LIN {X 0,Y 213.734,Z 203.361,A -85,B 0,C 180,E1 -20828.664,E2 -20828.664} C_VEL
LIN {X 0,Y 213.771,Z 203.358,A -85,B 0,C 180,E1 -20833.676,E2 -20833.676} C_VEL
LIN {X 0,Y 213.726,Z 203.362,A -85,B 0,C 180,E1 -20836.337,E2 -20836.337} C_VEL
LIN {X 0,Y 213.733,Z 203.362,A -85,B 0,C 180,E1 -20841.337,E2 -20841.337} C_VEL
LIN {X 0,Y 213.765,Z 203.356,A -85,B 0,C 180,E1 -20846.021,E2 -20846.021} C_VEL
LIN {X 0,Y 213.777,Z 203.356,A -85,B 0,C 180,E1 -20850.455,E2 -20850.455} C_VEL
LIN {X 0,Y 213.798,Z 203.348,A -85,B 0,C 180,E1 -20854.702,E2 -20854.702} C_VEL
LIN {X 0,Y 213.809,Z 203.349,A -85,B 0,C 180,E1 -20858.804,E2 -20858.804} C_VEL
LIN {X 0,Y 213.94,Z 203.337,A -85,B 0,C 180,E1 -20862.804,E2 -20862.804} C_VEL
LIN {X 0,Y 213.95,Z 203.333,A -85,B 0,C 180,E1 -20866.707,E2 -20866.707} C_VEL
LIN {X 0,Y 214.139,Z 203.305,A -85,B 0,C 180,E1 -20870.556,E2 -20870.556} C_VEL
LIN {X 0,Y 214.096,Z 203.312,A -85,B 0,C 180,E1 -20874.349,E2 -20874.349} C_VEL
LIN {X 0,Y 214.441,Z 203.245,A -85,B 0,C 180,E1 -20878.123,E2 -20878.123} C_VEL
LIN {X 0,Y 214.547,Z 203.245,A -85,B 0,C 180,E1 -20880.001,E2 -20880.001} C_VEL
LIN {X 0,Y 214.442,Z 203.27,A -85,B 0,C 180,E1 -20881.879,E2 -20881.879} C_VEL
LIN {X 0,Y 214.196,Z 203.304,A -85,B 0,C 180,E1 -20887.543,E2 -20887.543} C_VEL
LIN {X 0,Y 213.997,Z 203.329,A -85,B 0,C 180,E1 -20891.365,E2 -20891.365} C_VEL
LIN {X 0,Y 213.931,Z 203.337,A -85,B 0,C 180,E1 -20895.238,E2 -20895.238} C_VEL
LIN {X 0,Y 213.839,Z 203.349,A -85,B 0,C 180,E1 -20899.188,E2 -20899.188} C_VEL
LIN {X 0,Y 213.847,Z 203.35,A -85,B 0,C 180,E1 -20903.228,E2 -20903.228} C_VEL
LIN {X 0,Y 213.862,Z 203.711,A -85,B 0,C 180,E1 -20907.393,E2 -20907.393} C_VEL
LIN {X 0,Y 214.057,Z 205.405,A -85,B 0,C 180,E1 -20911.691,E2 -20911.691} C_VEL
LIN {X 0,Y 214.298,Z 207.41,A -85,B 0,C 180,E1 -20916.181,E2 -20916.181} C_VEL
LIN {X 0,Y 214.668,Z 209.889,A -85,B 0,C 180,E1 -20921.15,E2 -20921.15} C_VEL
LIN {X 0,Y 214.851,Z 211.419,A -85,B 0,C 180,E1 -20923.976,E2 -20923.976} C_VEL
LIN {X 0,Y 214.879,Z 212.962,A -85,B 0,C 180,E1 -20926.62,E2 -20926.62} C_VEL
LIN {X 0,Y 214.729,Z 214.501,A -85,B 0,C 180,E1 -20929.112,E2 -20929.112} C_VEL
LIN {X 0,Y 213.905,Z 217.533,A -85,B 0,C 180,E1 -20933.744,E2 -20933.744} C_VEL
LIN {X 0,Y 213.736,Z 218.183,A -85,B 0,C 180,E1 -20934.657,E2 -20934.657} C_VEL
LIN {X 0,Y 214.709,Z 221.629,A -85,B 0,C 180,E1 -20935.032,E2 -20935.032} C_VEL
LIN {X 0,Y 218.172,Z 231.953,A -85,B 0,C 180,E1 -20936.447,E2 -20936.447} C_VEL
LIN {X 0,Y 221.362,Z 245.09,A -85,B 0,C 180,E1 -20938.386,E2 -20938.386} C_VEL
LIN {X 0,Y 223.043,Z 255.539,A -85,B 0,C 180,E1 -20940.087,E2 -20940.087} C_VEL
LIN {X 0,Y 223.802,Z 263.81,A -85,B 0,C 180,E1 -20941.557,E2 -20941.557} C_VEL
LIN {X 0,Y 223.987,Z 273.301,A -85,B 0,C 180,E1 -20943.443,E2 -20943.443} C_VEL
LIN {X 0,Y 223.651,Z 277.858,A -85,B 0,C 180,E1 -20944.401,E2 -20944.401} C_VEL
LIN {X 0,Y 220.772,Z 288.296,A -85,B 0,C 180,E1 -20946.813,E2 -20946.813} C_VEL
LIN {X 0,Y 218.78,Z 295.491,A -85,B 0,C 180,E1 -20948.892,E2 -20948.892} C_VEL
LIN {X 0,Y 216.831,Z 301.814,A -85,B 0,C 180,E1 -20951.088,E2 -20951.088} C_VEL
LIN {X 0,Y 215.383,Z 306.725,A -85,B 0,C 180,E1 -20953.129,E2 -20953.129} C_VEL
LIN {X 0,Y 213.86,Z 309.596,A -85,B 0,C 180,E1 -20954.466,E2 -20954.466} C_VEL
LIN {X 0,Y 209.854,Z 313.608,A -85,B 0,C 180,E1 -20956.656,E2 -20956.656} C_VEL
LIN {X 0,Y 206.095,Z 317.034,A -85,B 0,C 180,E1 -20959.002,E2 -20959.002} C_VEL
LIN {X 0,Y 204.99,Z 318.689,A -85,B 0,C 180,E1 -20960.554,E2 -20960.554} C_VEL
LIN {X 0,Y 204.442,Z 321.502,A -85,B 0,C 180,E1 -20964.081,E2 -20964.081} C_VEL
LIN {X 0,Y 204.339,Z 322.566,A -85,B 0,C 180,E1 -20966.056,E2 -20966.056} C_VEL
LIN {X 0,Y 204.365,Z 323.161,A -85,B 0,C 180,E1 -20968.029,E2 -20968.029} C_VEL
LIN {X 0,Y 204.429,Z 323.319,A -85,B 0,C 180,E1 -20970,E2 -20970} C_VEL
LIN {X 0,Y 204.366,Z 323.161,A -85,B 0,C 180,E1 -20971.971,E2 -20971.971} C_VEL
LIN {X 0,Y 204.36,Z 322.491,A -85,B 0,C 180,E1 -20974.184,E2 -20974.184} C_VEL
LIN {X 0,Y 204.675,Z 320.109,A -85,B 0,C 180,E1 -20977.894,E2 -20977.894} C_VEL
LIN {X 0,Y 205.363,Z 317.152,A -85,B 0,C 180,E1 -20980.849,E2 -20980.849} C_VEL
LIN {X 0,Y 206.412,Z 313.156,A -85,B 0,C 180,E1 -20983.788,E2 -20983.788} C_VEL
LIN {X 0,Y 208.044,Z 308.023,A -85,B 0,C 180,E1 -20986.687,E2 -20986.687} C_VEL
LIN {X 0,Y 209.717,Z 302.758,A -85,B 0,C 180,E1 -20989.071,E2 -20989.071} C_VEL
LIN {X 0,Y 211.811,Z 296.441,A -85,B 0,C 180,E1 -20991.406,E2 -20991.406} C_VEL
LIN {X 0,Y 213.493,Z 290.484,A -85,B 0,C 180,E1 -20993.267,E2 -20993.267} C_VEL
LIN {X 0,Y 215.527,Z 283.556,A -85,B 0,C 180,E1 -20995.081,E2 -20995.081} C_VEL
LIN {X 0,Y 217.216,Z 277.645,A -85,B 0,C 180,E1 -20996.415,E2 -20996.415} C_VEL
LIN {X 0,Y 217.345,Z 267.824,A -85,B 0,C 180,E1 -20998.547,E2 -20998.547} C_VEL
LIN {X 0,Y 216.74,Z 258.58,A -85,B 0,C 180,E1 -21000.341,E2 -21000.341} C_VEL
LIN {X 0,Y 215.465,Z 249.191,A -85,B 0,C 180,E1 -21001.997,E2 -21001.997} C_VEL
LIN {X 0,Y 213.303,Z 238.611,A -85,B 0,C 180,E1 -21003.699,E2 -21003.699} C_VEL
LIN {X 0,Y 210.592,Z 229.072,A -85,B 0,C 180,E1 -21005.149,E2 -21005.149} C_VEL
LIN {X 0,Y 207.683,Z 220.968,A -85,B 0,C 180,E1 -21006.358,E2 -21006.358} C_VEL
LIN {X 0,Y 206.902,Z 217.966,A -85,B 0,C 180,E1 -21006.726,E2 -21006.726} C_VEL
LIN {X 0,Y 207.478,Z 215.775,A -85,B 0,C 180,E1 -21010.06,E2 -21010.06} C_VEL
LIN {X 0,Y 207.75,Z 214.247,A -85,B 0,C 180,E1 -21012.576,E2 -21012.576} C_VEL
LIN {X 0,Y 207.807,Z 212.729,A -85,B 0,C 180,E1 -21015.252,E2 -21015.252} C_VEL
LIN {X 0,Y 207.52,Z 210.25,A -85,B 0,C 180,E1 -21019.948,E2 -21019.948} C_VEL
LIN {X 0,Y 207.225,Z 207.973,A -85,B 0,C 180,E1 -21024.79,E2 -21024.79} C_VEL
LIN {X 0,Y 206.981,Z 206.053,A -85,B 0,C 180,E1 -21029.38,E2 -21029.38} C_VEL
LIN {X 0,Y 206.751,Z 204.425,A -85,B 0,C 180,E1 -21033.774,E2 -21033.774} C_VEL
LIN {X 0,Y 206.757,Z 204.236,A -85,B 0,C 180,E1 -21038.042,E2 -21038.042} C_VEL
LIN {X 0,Y 206.873,Z 204.219,A -85,B 0,C 180,E1 -21042.195,E2 -21042.195} C_VEL
LIN {X 0,Y 206.893,Z 204.215,A -85,B 0,C 180,E1 -21046.243,E2 -21046.243} C_VEL
LIN {X 0,Y 207.098,Z 204.19,A -85,B 0,C 180,E1 -21050.23,E2 -21050.23} C_VEL
LIN {X 0,Y 207.058,Z 204.194,A -85,B 0,C 180,E1 -21054.155,E2 -21054.155} C_VEL
LIN {X 0,Y 207.378,Z 204.15,A -85,B 0,C 180,E1 -21058.057,E2 -21058.057} C_VEL
LIN {X 0,Y 207.512,Z 204.12,A -85,B 0,C 180,E1 -21059.999,E2 -21059.999} C_VEL
LIN {X 0,Y 207.378,Z 204.124,A -85,B 0,C 180,E1 -21061.941,E2 -21061.941} C_VEL
LIN {X 0,Y 207.138,Z 204.182,A -85,B 0,C 180,E1 -21067.799,E2 -21067.799} C_VEL
LIN {X 0,Y 206.928,Z 204.21,A -85,B 0,C 180,E1 -21071.757,E2 -21071.757} C_VEL
LIN {X 0,Y 206.863,Z 204.214,A -85,B 0,C 180,E1 -21075.77,E2 -21075.77} C_VEL
LIN {X 0,Y 206.78,Z 204.219,A -85,B 0,C 180,E1 -21079.868,E2 -21079.868} C_VEL
LIN {X 0,Y 206.76,Z 204.227,A -85,B 0,C 180,E1 -21084.071,E2 -21084.071} C_VEL
LIN {X 0,Y 206.741,Z 204.233,A -85,B 0,C 180,E1 -21088.418,E2 -21088.418} C_VEL
LIN {X 0,Y 206.705,Z 204.236,A -85,B 0,C 180,E1 -21092.955,E2 -21092.955} C_VEL
LIN {X 0,Y 206.718,Z 204.234,A -85,B 0,C 180,E1 -21095.32,E2 -21095.32} C_VEL
LIN {X 0,Y 206.667,Z 204.242,A -85,B 0,C 180,E1 -21100.248,E2 -21100.248} C_VEL
LIN {X 0,Y 206.645,Z 204.245,A -85,B 0,C 180,E1 -21104.422,E2 -21104.422} C_VEL
LIN {X 0,Y 206.659,Z 204.241,A -85,B 0,C 180,E1 -21109.749,E2 -21109.749} C_VEL
LIN {X 0,Y 206.695,Z 204.302,A -85,B 0,C 180,E1 -21113.054,E2 -21113.054} C_VEL
LIN {X 0,Y 207.675,Z 207.027,A -85,B 0,C 180,E1 -21113.414,E2 -21113.414} C_VEL
LIN {X 0,Y 209.169,Z 209.299,A -85,B 0,C 180,E1 -21113.848,E2 -21113.848} C_VEL
LIN {X 0,Y 214.287,Z 218.562,A -85,B 0,C 180,E1 -21115.53,E2 -21115.53} C_VEL
LIN {X 0,Y 219.411,Z 229.769,A -85,B 0,C 180,E1 -21117.559,E2 -21117.559} C_VEL
LIN {X 0,Y 223.293,Z 240.321,A -85,B 0,C 180,E1 -21119.548,E2 -21119.548} C_VEL
LIN {X 0,Y 226.869,Z 250.975,A -85,B 0,C 180,E1 -21121.781,E2 -21121.781} C_VEL
LIN {X 0,Y 230.64,Z 259.099,A -85,B 0,C 180,E1 -21123.821,E2 -21123.821} C_VEL
LIN {X 0,Y 235.944,Z 267.711,A -85,B 0,C 180,E1 -21126.336,E2 -21126.336} C_VEL
LIN {X 0,Y 242.815,Z 276.218,A -85,B 0,C 180,E1 -21129.203,E2 -21129.203} C_VEL
LIN {X 0,Y 250.96,Z 283.988,A -85,B 0,C 180,E1 -21132.201,E2 -21132.201} C_VEL
LIN {X 0,Y 258.511,Z 290.027,A -85,B 0,C 180,E1 -21134.816,E2 -21134.816} C_VEL
LIN {X 0,Y 267.698,Z 296.215,A -85,B 0,C 180,E1 -21137.876,E2 -21137.876} C_VEL
LIN {X 0,Y 274.849,Z 300.626,A -85,B 0,C 180,E1 -21140.433,E2 -21140.433} C_VEL
LIN {X 0,Y 280.845,Z 303.994,A -85,B 0,C 180,E1 -21142.812,E2 -21142.812} C_VEL
LIN {X 0,Y 283.79,Z 305.702,A -85,B 0,C 180,E1 -21144.315,E2 -21144.315} C_VEL
LIN {X 0,Y 285.961,Z 307.015,A -85,B 0,C 180,E1 -21145.772,E2 -21145.772} C_VEL
LIN {X 0,Y 288.415,Z 308.115,A -85,B 0,C 180,E1 -21147.514,E2 -21147.514} C_VEL
LIN {X 0,Y 289.581,Z 308.494,A -85,B 0,C 180,E1 -21148.609,E2 -21148.609} C_VEL
LIN {X 0,Y 290.591,Z 308.662,A -85,B 0,C 180,E1 -21150,E2 -21150} C_VEL
LIN {X 0,Y 289.596,Z 308.494,A -85,B 0,C 180,E1 -21151.391,E2 -21151.391} C_VEL
LIN {X 0,Y 287.978,Z 307.95,A -85,B 0,C 180,E1 -21152.798,E2 -21152.798} C_VEL
LIN {X 0,Y 285.97,Z 307.014,A -85,B 0,C 180,E1 -21154.228,E2 -21154.228} C_VEL
LIN {X 0,Y 282.805,Z 305.083,A -85,B 0,C 180,E1 -21156.266,E2 -21156.266} C_VEL
LIN {X 0,Y 280.814,Z 303.995,A -85,B 0,C 180,E1 -21157.189,E2 -21157.189} C_VEL
LIN {X 0,Y 274.935,Z 300.623,A -85,B 0,C 180,E1 -21159.564,E2 -21159.564} C_VEL
LIN {X 0,Y 267.713,Z 296.215,A -85,B 0,C 180,E1 -21162.123,E2 -21162.123} C_VEL
LIN {X 0,Y 258.512,Z 290.025,A -85,B 0,C 180,E1 -21165.185,E2 -21165.185} C_VEL
LIN {X 0,Y 250.459,Z 283.545,A -85,B 0,C 180,E1 -21167.978,E2 -21167.978} C_VEL
LIN {X 0,Y 242.837,Z 276.198,A -85,B 0,C 180,E1 -21170.8,E2 -21170.8} C_VEL
LIN {X 0,Y 235.921,Z 267.776,A -85,B 0,C 180,E1 -21173.651,E2 -21173.651} C_VEL
LIN {X 0,Y 230.036,Z 257.992,A -85,B 0,C 180,E1 -21176.481,E2 -21176.481} C_VEL
LIN {X 0,Y 225.736,Z 248.075,A -85,B 0,C 180,E1 -21178.874,E2 -21178.874} C_VEL
LIN {X 0,Y 222.35,Z 237.621,A -85,B 0,C 180,E1 -21180.963,E2 -21180.963} C_VEL
LIN {X 0,Y 219.407,Z 229.775,A -85,B 0,C 180,E1 -21182.441,E2 -21182.441} C_VEL
LIN {X 0,Y 214.208,Z 218.418,A -85,B 0,C 180,E1 -21184.497,E2 -21184.497} C_VEL
LIN {X 0,Y 208.571,Z 208.219,A -85,B 0,C 180,E1 -21186.356,E2 -21186.356} C_VEL
LIN {X 0,Y 207.015,Z 205.604,A -85,B 0,C 180,E1 -21186.82,E2 -21186.82} C_VEL
LIN {X 0,Y 206.689,Z 204.239,A -85,B 0,C 180,E1 -21187.018,E2 -21187.018} C_VEL
LIN {X 0,Y 206.675,Z 204.242,A -85,B 0,C 180,E1 -21191.575,E2 -21191.575} C_VEL
LIN {X 0,Y 206.648,Z 204.244,A -85,B 0,C 180,E1 -21195.577,E2 -21195.577} C_VEL
LIN {X 0,Y 206.667,Z 204.242,A -85,B 0,C 180,E1 -21199.752,E2 -21199.752} C_VEL
LIN {X 0,Y 206.728,Z 204.233,A -85,B 0,C 180,E1 -21204.696,E2 -21204.696} C_VEL
LIN {X 0,Y 206.72,Z 204.235,A -85,B 0,C 180,E1 -21209.34,E2 -21209.34} C_VEL
LIN {X 0,Y 206.729,Z 204.23,A -85,B 0,C 180,E1 -21213.773,E2 -21213.773} C_VEL
LIN {X 0,Y 206.754,Z 204.23,A -85,B 0,C 180,E1 -21218.044,E2 -21218.044} C_VEL
LIN {X 0,Y 206.87,Z 204.216,A -85,B 0,C 180,E1 -21222.197,E2 -21222.197} C_VEL
LIN {X 0,Y 206.892,Z 204.21,A -85,B 0,C 180,E1 -21226.245,E2 -21226.245} C_VEL
LIN {X 0,Y 207.097,Z 204.182,A -85,B 0,C 180,E1 -21230.232,E2 -21230.232} C_VEL
LIN {X 0,Y 207.058,Z 204.191,A -85,B 0,C 180,E1 -21234.157,E2 -21234.157} C_VEL
LIN {X 0,Y 207.378,Z 204.124,A -85,B 0,C 180,E1 -21238.059,E2 -21238.059} C_VEL
LIN {X 0,Y 207.512,Z 204.12,A -85,B 0,C 180,E1 -21240.001,E2 -21240.001} C_VEL
LIN {X 0,Y 207.378,Z 204.15,A -85,B 0,C 180,E1 -21241.943,E2 -21241.943} C_VEL
LIN {X 0,Y 207.138,Z 204.184,A -85,B 0,C 180,E1 -21247.801,E2 -21247.801} C_VEL
LIN {X 0,Y 206.923,Z 204.212,A -85,B 0,C 180,E1 -21251.76,E2 -21251.76} C_VEL
LIN {X 0,Y 206.865,Z 204.219,A -85,B 0,C 180,E1 -21255.772,E2 -21255.772} C_VEL
LIN {X 0,Y 206.783,Z 204.229,A -85,B 0,C 180,E1 -21259.87,E2 -21259.87} C_VEL
LIN {X 0,Y 206.763,Z 204.231,A -85,B 0,C 180,E1 -21264.073,E2 -21264.073} C_VEL
LIN {X 0,Y 206.751,Z 204.419,A -85,B 0,C 180,E1 -21266.226,E2 -21266.226} C_VEL
LIN {X 0,Y 206.981,Z 206.052,A -85,B 0,C 180,E1 -21270.62,E2 -21270.62} C_VEL
LIN {X 0,Y 207.238,Z 208.124,A -85,B 0,C 180,E1 -21275.522,E2 -21275.522} C_VEL
LIN {X 0,Y 207.526,Z 210.283,A -85,B 0,C 180,E1 -21280.051,E2 -21280.051} C_VEL
LIN {X 0,Y 207.807,Z 212.733,A -85,B 0,C 180,E1 -21284.748,E2 -21284.748} C_VEL
LIN {X 0,Y 207.711,Z 214.682,A -85,B 0,C 180,E1 -21288.107,E2 -21288.107} C_VEL
LIN {X 0,Y 207.066,Z 217.312,A -85,B 0,C 180,E1 -21292.344,E2 -21292.344} C_VEL
LIN {X 0,Y 206.902,Z 217.945,A -85,B 0,C 180,E1 -21293.274,E2 -21293.274} C_VEL
LIN {X 0,Y 207.941,Z 221.513,A -85,B 0,C 180,E1 -21293.725,E2 -21293.725} C_VEL
LIN {X 0,Y 211.686,Z 232.468,A -85,B 0,C 180,E1 -21295.342,E2 -21295.342} C_VEL
LIN {X 0,Y 214.502,Z 243.922,A -85,B 0,C 180,E1 -21297.124,E2 -21297.124} C_VEL
LIN {X 0,Y 216.346,Z 255.133,A -85,B 0,C 180,E1 -21299.033,E2 -21299.033} C_VEL
LIN {X 0,Y 217.135,Z 263.358,A -85,B 0,C 180,E1 -21300.556,E2 -21300.556} C_VEL
LIN {X 0,Y 217.327,Z 272.309,A -85,B 0,C 180,E1 -21302.387,E2 -21302.387} C_VEL
LIN {X 0,Y 217.206,Z 277.645,A -85,B 0,C 180,E1 -21303.583,E2 -21303.583} C_VEL
LIN {X 0,Y 214.502,Z 287.229,A -85,B 0,C 180,E1 -21305.824,E2 -21305.824} C_VEL
LIN {X 0,Y 212.22,Z 294.76,A -85,B 0,C 180,E1 -21308.015,E2 -21308.015} C_VEL
LIN {X 0,Y 210.107,Z 301.602,A -85,B 0,C 180,E1 -21310.458,E2 -21310.458} C_VEL
LIN {X 0,Y 208.453,Z 306.868,A -85,B 0,C 180,E1 -21312.738,E2 -21312.738} C_VEL
LIN {X 0,Y 206.894,Z 311.601,A -85,B 0,C 180,E1 -21315.24,E2 -21315.24} C_VEL
LIN {X 0,Y 205.684,Z 315.933,A -85,B 0,C 180,E1 -21318.17,E2 -21318.17} C_VEL
LIN {X 0,Y 204.99,Z 318.689,A -85,B 0,C 180,E1 -21320.554,E2 -21320.554} C_VEL
LIN {X 0,Y 203.994,Z 320.173,A -85,B 0,C 180,E1 -21322.141,E2 -21322.141} C_VEL
LIN {X 0,Y 200.83,Z 321.86,A -85,B 0,C 180,E1 -21324.759,E2 -21324.759} C_VEL
LIN {X 0,Y 198.343,Z 322.679,A -85,B 0,C 180,E1 -21326.924,E2 -21326.924} C_VEL
LIN {X 0,Y 197.287,Z 323.105,A -85,B 0,C 180,E1 -21328.908,E2 -21328.908} C_VEL
LIN {X 0,Y 197.278,Z 323.045,A -85,B 0,C 180,E1 -21329.195,E2 -21329.195} C_VEL
LIN {X 0,Y 197.271,Z 322.95,A -85,B 0,C 180,E1 -21332.042,E2 -21332.042} C_VEL
LIN {X 0,Y 197.257,Z 322.355,A -85,B 0,C 180,E1 -21334.086,E2 -21334.086} C_VEL
LIN {X 0,Y 197.642,Z 319.897,A -85,B 0,C 180,E1 -21338.177,E2 -21338.177} C_VEL
LIN {X 0,Y 198.355,Z 316.94,A -85,B 0,C 180,E1 -21341.237,E2 -21341.237} C_VEL
LIN {X 0,Y 199.482,Z 312.944,A -85,B 0,C 180,E1 -21344.277,E2 -21344.277} C_VEL
LIN {X 0,Y 201.225,Z 307.811,A -85,B 0,C 180,E1 -21347.269,E2 -21347.269} C_VEL
LIN {X 0,Y 202.991,Z 302.546,A -85,B 0,C 180,E1 -21349.728,E2 -21349.728} C_VEL
LIN {X 0,Y 204.751,Z 297.606,A -85,B 0,C 180,E1 -21351.653,E2 -21351.653} C_VEL
LIN {X 0,Y 206.953,Z 290.271,A -85,B 0,C 180,E1 -21354.048,E2 -21354.048} C_VEL
LIN {X 0,Y 209.092,Z 283.344,A -85,B 0,C 180,E1 -21355.909,E2 -21355.909} C_VEL
LIN {X 0,Y 210.553,Z 278.522,A -85,B 0,C 180,E1 -21357.051,E2 -21357.051} C_VEL
LIN {X 0,Y 210.739,Z 267.6,A -85,B 0,C 180,E1 -21359.528,E2 -21359.528} C_VEL
LIN {X 0,Y 210.227,Z 259.06,A -85,B 0,C 180,E1 -21361.265,E2 -21361.265} C_VEL
LIN {X 0,Y 208.917,Z 249.242,A -85,B 0,C 180,E1 -21363.086,E2 -21363.086} C_VEL
LIN {X 0,Y 206.806,Z 239.117,A -85,B 0,C 180,E1 -21364.823,E2 -21364.823} C_VEL
LIN {X 0,Y 203.969,Z 229.166,A -85,B 0,C 180,E1 -21366.44,E2 -21366.44} C_VEL
LIN {X 0,Y 201.107,Z 221.229,A -85,B 0,C 180,E1 -21367.719,E2 -21367.719} C_VEL
LIN {X 0,Y 200.134,Z 218.248,A -85,B 0,C 180,E1 -21368.111,E2 -21368.111} C_VEL
LIN {X 0,Y 200.126,Z 217.72,A -85,B 0,C 180,E1 -21368.233,E2 -21368.233} C_VEL
LIN {X 0,Y 200.695,Z 215.02,A -85,B 0,C 180,E1 -21372.659,E2 -21372.659} C_VEL
LIN {X 0,Y 200.725,Z 213.424,A -85,B 0,C 180,E1 -21375.551,E2 -21375.551} C_VEL
LIN {X 0,Y 200.61,Z 212.027,A -85,B 0,C 180,E1 -21378.268,E2 -21378.268} C_VEL
LIN {X 0,Y 200.229,Z 209.62,A -85,B 0,C 180,E1 -21383.365,E2 -21383.365} C_VEL
LIN {X 0,Y 200.004,Z 207.585,A -85,B 0,C 180,E1 -21388.19,E2 -21388.19} C_VEL
LIN {X 0,Y 199.782,Z 205.885,A -85,B 0,C 180,E1 -21392.785,E2 -21392.785} C_VEL
LIN {X 0,Y 199.68,Z 205.141,A -85,B 0,C 180,E1 -21395.015,E2 -21395.015} C_VEL
LIN {X 0,Y 199.7,Z 205.114,A -85,B 0,C 180,E1 -21399.394,E2 -21399.394} C_VEL
LIN {X 0,Y 199.803,Z 205.098,A -85,B 0,C 180,E1 -21403.655,E2 -21403.655} C_VEL
LIN {X 0,Y 199.873,Z 205.089,A -85,B 0,C 180,E1 -21407.819,E2 -21407.819} C_VEL
LIN {X 0,Y 200.087,Z 205.063,A -85,B 0,C 180,E1 -21411.922,E2 -21411.922} C_VEL
LIN {X 0,Y 200.318,Z 205.03,A -85,B 0,C 180,E1 -21417.988,E2 -21417.988} C_VEL
LIN {X 0,Y 200.476,Z 204.996,A -85,B 0,C 180,E1 -21419.999,E2 -21419.999} C_VEL
LIN {X 0,Y 200.022,Z 205.051,A -85,B 0,C 180,E1 -21424.029,E2 -21424.029} C_VEL
LIN {X 0,Y 200.086,Z 205.059,A -85,B 0,C 180,E1 -21428.076,E2 -21428.076} C_VEL
LIN {X 0,Y 199.876,Z 205.087,A -85,B 0,C 180,E1 -21432.178,E2 -21432.178} C_VEL
LIN {X 0,Y 199.801,Z 205.094,A -85,B 0,C 180,E1 -21436.343,E2 -21436.343} C_VEL
LIN {X 0,Y 199.697,Z 205.102,A -85,B 0,C 180,E1 -21440.604,E2 -21440.604} C_VEL
LIN {X 0,Y 199.669,Z 205.107,A -85,B 0,C 180,E1 -21444.984,E2 -21444.984} C_VEL
LIN {X 0,Y 199.671,Z 205.113,A -85,B 0,C 180,E1 -21449.521,E2 -21449.521} C_VEL
LIN {X 0,Y 199.66,Z 205.115,A -85,B 0,C 180,E1 -21452.352,E2 -21452.352} C_VEL
LIN {X 0,Y 199.636,Z 205.119,A -85,B 0,C 180,E1 -21456.759,E2 -21456.759} C_VEL
LIN {X 0,Y 199.636,Z 205.117,A -85,B 0,C 180,E1 -21459.32,E2 -21459.32} C_VEL
LIN {X 0,Y 199.586,Z 205.124,A -85,B 0,C 180,E1 -21462.315,E2 -21462.315} C_VEL
LIN {X 0,Y 199.584,Z 205.122,A -85,B 0,C 180,E1 -21465.231,E2 -21465.231} C_VEL
LIN {X 0,Y 199.637,Z 205.118,A -85,B 0,C 180,E1 -21470.757,E2 -21470.757} C_VEL
LIN {X 0,Y 199.665,Z 205.115,A -85,B 0,C 180,E1 -21471.535,E2 -21471.535} C_VEL
LIN {X 0,Y 200.686,Z 208.007,A -85,B 0,C 180,E1 -21471.961,E2 -21471.961} C_VEL
LIN {X 0,Y 202.276,Z 210.36,A -85,B 0,C 180,E1 -21472.456,E2 -21472.456} C_VEL
LIN {X 0,Y 207.913,Z 220.424,A -85,B 0,C 180,E1 -21474.456,E2 -21474.456} C_VEL
LIN {X 0,Y 213.644,Z 233.269,A -85,B 0,C 180,E1 -21476.975,E2 -21476.975} C_VEL
LIN {X 0,Y 217.186,Z 243.33,A -85,B 0,C 180,E1 -21479.036,E2 -21479.036} C_VEL
LIN {X 0,Y 220.118,Z 252.755,A -85,B 0,C 180,E1 -21481.132,E2 -21481.132} C_VEL
LIN {X 0,Y 223.373,Z 260.472,A -85,B 0,C 180,E1 -21483.146,E2 -21483.146} C_VEL
LIN {X 0,Y 228.444,Z 269.262,A -85,B 0,C 180,E1 -21485.839,E2 -21485.839} C_VEL
LIN {X 0,Y 234.196,Z 276.747,A -85,B 0,C 180,E1 -21488.476,E2 -21488.476} C_VEL
LIN {X 0,Y 241.181,Z 283.829,A -85,B 0,C 180,E1 -21491.305,E2 -21491.305} C_VEL
LIN {X 0,Y 248.557,Z 289.853,A -85,B 0,C 180,E1 -21494.016,E2 -21494.016} C_VEL
LIN {X 0,Y 256.024,Z 295.018,A -85,B 0,C 180,E1 -21496.629,E2 -21496.629} C_VEL
LIN {X 0,Y 263.684,Z 299.525,A -85,B 0,C 180,E1 -21499.247,E2 -21499.247} C_VEL
LIN {X 0,Y 269.969,Z 302.954,A -85,B 0,C 180,E1 -21501.58,E2 -21501.58} C_VEL
LIN {X 0,Y 275.623,Z 305.739,A -85,B 0,C 180,E1 -21503.949,E2 -21503.949} C_VEL
LIN {X 0,Y 278.411,Z 307.238,A -85,B 0,C 180,E1 -21505.657,E2 -21505.657} C_VEL
LIN {X 0,Y 281.34,Z 308.428,A -85,B 0,C 180,E1 -21507.711,E2 -21507.711} C_VEL
LIN {X 0,Y 282.29,Z 308.71,A -85,B 0,C 180,E1 -21508.573,E2 -21508.573} C_VEL
LIN {X 0,Y 283.424,Z 308.872,A -85,B 0,C 180,E1 -21510,E2 -21510} C_VEL
LIN {X 0,Y 282.302,Z 308.71,A -85,B 0,C 180,E1 -21511.427,E2 -21511.427} C_VEL
LIN {X 0,Y 280.506,Z 308.174,A -85,B 0,C 180,E1 -21512.872,E2 -21512.872} C_VEL
LIN {X 0,Y 278.414,Z 307.238,A -85,B 0,C 180,E1 -21514.343,E2 -21514.343} C_VEL
LIN {X 0,Y 275.62,Z 305.746,A -85,B 0,C 180,E1 -21516.045,E2 -21516.045} C_VEL
LIN {X 0,Y 269.976,Z 302.939,A -85,B 0,C 180,E1 -21518.429,E2 -21518.429} C_VEL
LIN {X 0,Y 263.7,Z 299.525,A -85,B 0,C 180,E1 -21520.752,E2 -21520.752} C_VEL
LIN {X 0,Y 256.041,Z 295.013,A -85,B 0,C 180,E1 -21523.372,E2 -21523.372} C_VEL
LIN {X 0,Y 246.957,Z 288.711,A -85,B 0,C 180,E1 -21526.534,E2 -21526.534} C_VEL
LIN {X 0,Y 237.617,Z 280.437,A -85,B 0,C 180,E1 -21530.108,E2 -21530.108} C_VEL
LIN {X 0,Y 230.919,Z 272.758,A -85,B 0,C 180,E1 -21532.983,E2 -21532.983} C_VEL
LIN {X 0,Y 225.807,Z 265.081,A -85,B 0,C 180,E1 -21535.501,E2 -21535.501} C_VEL
LIN {X 0,Y 222.091,Z 257.682,A -85,B 0,C 180,E1 -21537.621,E2 -21537.621} C_VEL
LIN {X 0,Y 218.717,Z 248.726,A -85,B 0,C 180,E1 -21539.823,E2 -21539.823} C_VEL
LIN {X 0,Y 215.491,Z 238.222,A -85,B 0,C 180,E1 -21542.012,E2 -21542.012} C_VEL
LIN {X 0,Y 211.714,Z 228.788,A -85,B 0,C 180,E1 -21543.914,E2 -21543.914} C_VEL
LIN {X 0,Y 207.267,Z 219.361,A -85,B 0,C 180,E1 -21545.765,E2 -21545.765} C_VEL
LIN {X 0,Y 203.029,Z 211.8,A -85,B 0,C 180,E1 -21547.295,E2 -21547.295} C_VEL
LIN {X 0,Y 201.489,Z 209.03,A -85,B 0,C 180,E1 -21547.818,E2 -21547.818} C_VEL
LIN {X 0,Y 200.01,Z 206.605,A -85,B 0,C 180,E1 -21548.297,E2 -21548.297} C_VEL
LIN {X 0,Y 199.679,Z 205.113,A -85,B 0,C 180,E1 -21548.504,E2 -21548.504} C_VEL
LIN {X 0,Y 199.616,Z 205.118,A -85,B 0,C 180,E1 -21552.325,E2 -21552.325} C_VEL
LIN {X 0,Y 199.604,Z 205.12,A -85,B 0,C 180,E1 -21555.237,E2 -21555.237} C_VEL
LIN {X 0,Y 199.636,Z 205.117,A -85,B 0,C 180,E1 -21560.68,E2 -21560.68} C_VEL
LIN {X 0,Y 199.631,Z 205.117,A -85,B 0,C 180,E1 -21565.719,E2 -21565.719} C_VEL
LIN {X 0,Y 199.7,Z 205.109,A -85,B 0,C 180,E1 -21568.138,E2 -21568.138} C_VEL
LIN {X 0,Y 199.684,Z 205.112,A -85,B 0,C 180,E1 -21572.773,E2 -21572.773} C_VEL
LIN {X 0,Y 199.735,Z 205.106,A -85,B 0,C 180,E1 -21577.23,E2 -21577.23} C_VEL
LIN {X 0,Y 199.793,Z 205.097,A -85,B 0,C 180,E1 -21581.759,E2 -21581.759} C_VEL
LIN {X 0,Y 199.832,Z 205.088,A -85,B 0,C 180,E1 -21585.749,E2 -21585.749} C_VEL
LIN {X 0,Y 200.02,Z 205.063,A -85,B 0,C 180,E1 -21589.883,E2 -21589.883} C_VEL
LIN {X 0,Y 200.019,Z 205.069,A -85,B 0,C 180,E1 -21593.95,E2 -21593.95} C_VEL
LIN {X 0,Y 200.317,Z 205.002,A -85,B 0,C 180,E1 -21597.991,E2 -21597.991} C_VEL
LIN {X 0,Y 200.476,Z 204.996,A -85,B 0,C 180,E1 -21600.001,E2 -21600.001} C_VEL
LIN {X 0,Y 200.024,Z 205.07,A -85,B 0,C 180,E1 -21604.031,E2 -21604.031} C_VEL
LIN {X 0,Y 200.087,Z 205.063,A -85,B 0,C 180,E1 -21608.078,E2 -21608.078} C_VEL
LIN {X 0,Y 199.873,Z 205.09,A -85,B 0,C 180,E1 -21612.181,E2 -21612.181} C_VEL
LIN {X 0,Y 199.803,Z 205.097,A -85,B 0,C 180,E1 -21616.345,E2 -21616.345} C_VEL
LIN {X 0,Y 199.7,Z 205.11,A -85,B 0,C 180,E1 -21620.606,E2 -21620.606} C_VEL
LIN {X 0,Y 199.68,Z 205.135,A -85,B 0,C 180,E1 -21624.985,E2 -21624.985} C_VEL
LIN {X 0,Y 199.892,Z 206.687,A -85,B 0,C 180,E1 -21629.488,E2 -21629.488} C_VEL
LIN {X 0,Y 200.112,Z 208.563,A -85,B 0,C 180,E1 -21634.19,E2 -21634.19} C_VEL
LIN {X 0,Y 200.445,Z 210.961,A -85,B 0,C 180,E1 -21639.525,E2 -21639.525} C_VEL
LIN {X 0,Y 200.656,Z 212.503,A -85,B 0,C 180,E1 -21642.649,E2 -21642.649} C_VEL
LIN {X 0,Y 200.735,Z 214.036,A -85,B 0,C 180,E1 -21645.556,E2 -21645.556} C_VEL
LIN {X 0,Y 200.612,Z 215.566,A -85,B 0,C 180,E1 -21648.271,E2 -21648.271} C_VEL
LIN {X 0,Y 200.086,Z 217.774,A -85,B 0,C 180,E1 -21651.848,E2 -21651.848} C_VEL
LIN {X 0,Y 200.976,Z 220.986,A -85,B 0,C 180,E1 -21652.237,E2 -21652.237} C_VEL
LIN {X 0,Y 201.858,Z 223.045,A -85,B 0,C 180,E1 -21652.578,E2 -21652.578} C_VEL
LIN {X 0,Y 205.739,Z 235.016,A -85,B 0,C 180,E1 -21654.5,E2 -21654.5} C_VEL
LIN {X 0,Y 208.18,Z 245.309,A -85,B 0,C 180,E1 -21656.223,E2 -21656.223} C_VEL
LIN {X 0,Y 209.754,Z 254.903,A -85,B 0,C 180,E1 -21657.946,E2 -21657.946} C_VEL
LIN {X 0,Y 210.592,Z 264.038,A -85,B 0,C 180,E1 -21659.729,E2 -21659.729} C_VEL
LIN {X 0,Y 210.754,Z 271.573,A -85,B 0,C 180,E1 -21661.326,E2 -21661.326} C_VEL
LIN {X 0,Y 210.549,Z 278.522,A -85,B 0,C 180,E1 -21662.949,E2 -21662.949} C_VEL
LIN {X 0,Y 208.031,Z 287.017,A -85,B 0,C 180,E1 -21665.021,E2 -21665.021} C_VEL
LIN {X 0,Y 205.429,Z 295.141,A -85,B 0,C 180,E1 -21667.477,E2 -21667.477} C_VEL
LIN {X 0,Y 203.418,Z 301.391,A -85,B 0,C 180,E1 -21669.788,E2 -21669.788} C_VEL
LIN {X 0,Y 201.952,Z 305.896,A -85,B 0,C 180,E1 -21671.748,E2 -21671.748} C_VEL
LIN {X 0,Y 200.019,Z 311.389,A -85,B 0,C 180,E1 -21674.721,E2 -21674.721} C_VEL
LIN {X 0,Y 198.697,Z 315.721,A -85,B 0,C 180,E1 -21677.748,E2 -21677.748} C_VEL
LIN {X 0,Y 197.909,Z 318.66,A -85,B 0,C 180,E1 -21680.422,E2 -21680.422} C_VEL
LIN {X 0,Y 197.369,Z 321.291,A -85,B 0,C 180,E1 -21683.868,E2 -21683.868} C_VEL
LIN {X 0,Y 197.247,Z 322.406,A -85,B 0,C 180,E1 -21686.088,E2 -21686.088} C_VEL
LIN {X 0,Y 197.278,Z 323.045,A -85,B 0,C 180,E1 -21689.195,E2 -21689.195} C_VEL
LIN {X 0,Y 196.641,Z 323.109,A -85,B 0,C 180,E1 -21690.897,E2 -21690.897} C_VEL
LIN {X 0,Y 195.046,Z 322.79,A -85,B 0,C 180,E1 -21692.568,E2 -21692.568} C_VEL
LIN {X 0,Y 191.389,Z 321.333,A -85,B 0,C 180,E1 -21695.934,E2 -21695.934} C_VEL
LIN {X 0,Y 190.513,Z 320.113,A -85,B 0,C 180,E1 -21697.976,E2 -21697.976} C_VEL
LIN {X 0,Y 190.544,Z 319.824,A -85,B 0,C 180,E1 -21698.271,E2 -21698.271} C_VEL
LIN {X 0,Y 191.362,Z 316.728,A -85,B 0,C 180,E1 -21701.653,E2 -21701.653} C_VEL
LIN {X 0,Y 192.573,Z 312.731,A -85,B 0,C 180,E1 -21704.801,E2 -21704.801} C_VEL
LIN {X 0,Y 194.434,Z 307.599,A -85,B 0,C 180,E1 -21707.893,E2 -21707.893} C_VEL
LIN {X 0,Y 196.306,Z 302.334,A -85,B 0,C 180,E1 -21710.43,E2 -21710.43} C_VEL
LIN {X 0,Y 198.114,Z 297.393,A -85,B 0,C 180,E1 -21712.417,E2 -21712.417} C_VEL
LIN {X 0,Y 200.46,Z 290.059,A -85,B 0,C 180,E1 -21714.879,E2 -21714.879} C_VEL
LIN {X 0,Y 202.722,Z 283.132,A -85,B 0,C 180,E1 -21716.787,E2 -21716.787} C_VEL
LIN {X 0,Y 204.001,Z 278.302,A -85,B 0,C 180,E1 -21717.994,E2 -21717.994} C_VEL
LIN {X 0,Y 204.243,Z 268.637,A -85,B 0,C 180,E1 -21720.302,E2 -21720.302} C_VEL
LIN {X 0,Y 203.626,Z 258.45,A -85,B 0,C 180,E1 -21722.467,E2 -21722.467} C_VEL
LIN {X 0,Y 202.462,Z 249.722,A -85,B 0,C 180,E1 -21724.179,E2 -21724.179} C_VEL
LIN {X 0,Y 200.199,Z 238.84,A -85,B 0,C 180,E1 -21726.154,E2 -21726.154} C_VEL
LIN {X 0,Y 197.263,Z 228.972,A -85,B 0,C 180,E1 -21727.886,E2 -21727.886} C_VEL
LIN {X 0,Y 194.446,Z 221.193,A -85,B 0,C 180,E1 -21729.239,E2 -21729.239} C_VEL
LIN {X 0,Y 193.348,Z 217.993,A -85,B 0,C 180,E1 -21729.706,E2 -21729.706} C_VEL
LIN {X 0,Y 193.292,Z 217.528,A -85,B 0,C 180,E1 -21729.793,E2 -21729.793} C_VEL
LIN {X 0,Y 193.653,Z 215.323,A -85,B 0,C 180,E1 -21733.593,E2 -21733.593} C_VEL
LIN {X 0,Y 193.633,Z 213.769,A -85,B 0,C 180,E1 -21736.544,E2 -21736.544} C_VEL
LIN {X 0,Y 193.442,Z 212.246,A -85,B 0,C 180,E1 -21739.724,E2 -21739.724} C_VEL
LIN {X 0,Y 193.139,Z 210.184,A -85,B 0,C 180,E1 -21744.392,E2 -21744.392} C_VEL
LIN {X 0,Y 192.919,Z 208.22,A -85,B 0,C 180,E1 -21749.334,E2 -21749.334} C_VEL
LIN {X 0,Y 192.837,Z 207.348,A -85,B 0,C 180,E1 -21751.718,E2 -21751.718} C_VEL
LIN {X 0,Y 192.706,Z 205.988,A -85,B 0,C 180,E1 -21756.347,E2 -21756.347} C_VEL
LIN {X 0,Y 192.731,Z 205.98,A -85,B 0,C 180,E1 -21761.456,E2 -21761.456} C_VEL
LIN {X 0,Y 192.762,Z 205.974,A -85,B 0,C 180,E1 -21765.212,E2 -21765.212} C_VEL
LIN {X 0,Y 192.944,Z 205.952,A -85,B 0,C 180,E1 -21769.565,E2 -21769.565} C_VEL
LIN {X 0,Y 192.982,Z 205.948,A -85,B 0,C 180,E1 -21773.727,E2 -21773.727} C_VEL
LIN {X 0,Y 193.259,Z 205.909,A -85,B 0,C 180,E1 -21777.915,E2 -21777.915} C_VEL
LIN {X 0,Y 193.44,Z 205.872,A -85,B 0,C 180,E1 -21779.999,E2 -21779.999} C_VEL
LIN {X 0,Y 192.968,Z 205.93,A -85,B 0,C 180,E1 -21784.176,E2 -21784.176} C_VEL
LIN {X 0,Y 193.033,Z 205.938,A -85,B 0,C 180,E1 -21788.373,E2 -21788.373} C_VEL
LIN {X 0,Y 192.802,Z 205.969,A -85,B 0,C 180,E1 -21792.632,E2 -21792.632} C_VEL
LIN {X 0,Y 192.754,Z 205.974,A -85,B 0,C 180,E1 -21796.958,E2 -21796.958} C_VEL
LIN {X 0,Y 192.633,Z 205.987,A -85,B 0,C 180,E1 -21801.396,E2 -21801.396} C_VEL
LIN {X 0,Y 192.661,Z 205.982,A -85,B 0,C 180,E1 -21804.224,E2 -21804.224} C_VEL
LIN {X 0,Y 192.647,Z 205.988,A -85,B 0,C 180,E1 -21808.891,E2 -21808.891} C_VEL
LIN {X 0,Y 192.597,Z 205.993,A -85,B 0,C 180,E1 -21813.185,E2 -21813.185} C_VEL
LIN {X 0,Y 192.606,Z 205.993,A -85,B 0,C 180,E1 -21816.607,E2 -21816.607} C_VEL
LIN {X 0,Y 192.527,Z 206.003,A -85,B 0,C 180,E1 -21821.075,E2 -21821.075} C_VEL
LIN {X 0,Y 192.513,Z 206.006,A -85,B 0,C 180,E1 -21826.083,E2 -21826.083} C_VEL
LIN {X 0,Y 192.548,Z 205.999,A -85,B 0,C 180,E1 -21829.874,E2 -21829.874} C_VEL
LIN {X 0,Y 193.549,Z 208.795,A -85,B 0,C 180,E1 -21830.322,E2 -21830.322} C_VEL
LIN {X 0,Y 195.391,Z 211.366,A -85,B 0,C 180,E1 -21830.934,E2 -21830.934} C_VEL
LIN {X 0,Y 201.537,Z 222.5,A -85,B 0,C 180,E1 -21833.325,E2 -21833.325} C_VEL
LIN {X 0,Y 206.507,Z 233.393,A -85,B 0,C 180,E1 -21835.66,E2 -21835.66} C_VEL
LIN {X 0,Y 210.258,Z 243.701,A -85,B 0,C 180,E1 -21837.921,E2 -21837.921} C_VEL
LIN {X 0,Y 212.912,Z 252.959,A -85,B 0,C 180,E1 -21840.05,E2 -21840.05} C_VEL
LIN {X 0,Y 215.793,Z 260.85,A -85,B 0,C 180,E1 -21842.153,E2 -21842.153} C_VEL
LIN {X 0,Y 220.264,Z 269.546,A -85,B 0,C 180,E1 -21844.887,E2 -21844.887} C_VEL
LIN {X 0,Y 225.277,Z 276.785,A -85,B 0,C 180,E1 -21847.505,E2 -21847.505} C_VEL
LIN {X 0,Y 232.022,Z 284.11,A -85,B 0,C 180,E1 -21850.538,E2 -21850.538} C_VEL
LIN {X 0,Y 238.826,Z 289.895,A -85,B 0,C 180,E1 -21853.248,E2 -21853.248} C_VEL
LIN {X 0,Y 246.284,Z 295.066,A -85,B 0,C 180,E1 -21855.98,E2 -21855.98} C_VEL
LIN {X 0,Y 254.55,Z 299.799,A -85,B 0,C 180,E1 -21858.857,E2 -21858.857} C_VEL
LIN {X 0,Y 259.535,Z 302.379,A -85,B 0,C 180,E1 -21860.65,E2 -21860.65} C_VEL
LIN {X 0,Y 264.018,Z 304.5,A -85,B 0,C 180,E1 -21862.352,E2 -21862.352} C_VEL
LIN {X 0,Y 268.426,Z 306.397,A -85,B 0,C 180,E1 -21864.216,E2 -21864.216} C_VEL
LIN {X 0,Y 270.759,Z 307.465,A -85,B 0,C 180,E1 -21865.534,E2 -21865.534} C_VEL
LIN {X 0,Y 274.268,Z 308.735,A -85,B 0,C 180,E1 -21867.921,E2 -21867.921} C_VEL
LIN {X 0,Y 276.245,Z 309.081,A -85,B 0,C 180,E1 -21870,E2 -21870} C_VEL
LIN {X 0,Y 274.999,Z 308.926,A -85,B 0,C 180,E1 -21871.464,E2 -21871.464} C_VEL
LIN {X 0,Y 272.99,Z 308.4,A -85,B 0,C 180,E1 -21872.951,E2 -21872.951} C_VEL
LIN {X 0,Y 270.753,Z 307.465,A -85,B 0,C 180,E1 -21874.466,E2 -21874.466} C_VEL
LIN {X 0,Y 267.846,Z 306.181,A -85,B 0,C 180,E1 -21876.025,E2 -21876.025} C_VEL
LIN {X 0,Y 262.708,Z 303.858,A -85,B 0,C 180,E1 -21878.185,E2 -21878.185} C_VEL
LIN {X 0,Y 257.103,Z 301.148,A -85,B 0,C 180,E1 -21880.245,E2 -21880.245} C_VEL
LIN {X 0,Y 249.039,Z 296.788,A -85,B 0,C 180,E1 -21883.048,E2 -21883.048} C_VEL
LIN {X 0,Y 241.125,Z 291.653,A -85,B 0,C 180,E1 -21885.883,E2 -21885.883} C_VEL
LIN {X 0,Y 233.776,Z 285.73,A -85,B 0,C 180,E1 -21888.747,E2 -21888.747} C_VEL
LIN {X 0,Y 226.658,Z 278.431,A -85,B 0,C 180,E1 -21891.844,E2 -21891.844} C_VEL
LIN {X 0,Y 221.619,Z 271.781,A -85,B 0,C 180,E1 -21894.346,E2 -21894.346} C_VEL
LIN {X 0,Y 218,Z 265.534,A -85,B 0,C 180,E1 -21896.438,E2 -21896.438} C_VEL
LIN {X 0,Y 214.298,Z 257.007,A -85,B 0,C 180,E1 -21898.91,E2 -21898.91} C_VEL
LIN {X 0,Y 211.834,Z 249.164,A -85,B 0,C 180,E1 -21900.86,E2 -21900.86} C_VEL
LIN {X 0,Y 208.76,Z 239.193,A -85,B 0,C 180,E1 -21903.067,E2 -21903.067} C_VEL
LIN {X 0,Y 204.527,Z 228.803,A -85,B 0,C 180,E1 -21905.306,E2 -21905.306} C_VEL
LIN {X 0,Y 199.919,Z 219.446,A -85,B 0,C 180,E1 -21907.312,E2 -21907.312} C_VEL
LIN {X 0,Y 194.503,Z 209.989,A -85,B 0,C 180,E1 -21909.385,E2 -21909.385} C_VEL
LIN {X 0,Y 192.961,Z 207.622,A -85,B 0,C 180,E1 -21909.926,E2 -21909.926} C_VEL
LIN {X 0,Y 192.559,Z 205.998,A -85,B 0,C 180,E1 -21910.148,E2 -21910.148} C_VEL
LIN {X 0,Y 192.544,Z 206.002,A -85,B 0,C 180,E1 -21913.908,E2 -21913.908} C_VEL
LIN {X 0,Y 192.527,Z 206.003,A -85,B 0,C 180,E1 -21918.925,E2 -21918.925} C_VEL
LIN {X 0,Y 192.606,Z 205.993,A -85,B 0,C 180,E1 -21923.393,E2 -21923.393} C_VEL
LIN {X 0,Y 192.604,Z 205.993,A -85,B 0,C 180,E1 -21927.06,E2 -21927.06} C_VEL
LIN {X 0,Y 192.661,Z 205.986,A -85,B 0,C 180,E1 -21931.693,E2 -21931.693} C_VEL
LIN {X 0,Y 192.702,Z 205.978,A -85,B 0,C 180,E1 -21936.349,E2 -21936.349} C_VEL
LIN {X 0,Y 192.729,Z 205.977,A -85,B 0,C 180,E1 -21941.459,E2 -21941.459} C_VEL
LIN {X 0,Y 192.761,Z 205.967,A -85,B 0,C 180,E1 -21945.215,E2 -21945.215} C_VEL
LIN {X 0,Y 192.942,Z 205.945,A -85,B 0,C 180,E1 -21949.568,E2 -21949.568} C_VEL
LIN {X 0,Y 192.982,Z 205.945,A -85,B 0,C 180,E1 -21953.729,E2 -21953.729} C_VEL
LIN {X 0,Y 193.259,Z 205.879,A -85,B 0,C 180,E1 -21957.917,E2 -21957.917} C_VEL
LIN {X 0,Y 193.44,Z 205.872,A -85,B 0,C 180,E1 -21960.001,E2 -21960.001} C_VEL
LIN {X 0,Y 192.969,Z 205.948,A -85,B 0,C 180,E1 -21964.178,E2 -21964.178} C_VEL
LIN {X 0,Y 193.034,Z 205.94,A -85,B 0,C 180,E1 -21968.375,E2 -21968.375} C_VEL
LIN {X 0,Y 192.8,Z 205.97,A -85,B 0,C 180,E1 -21972.635,E2 -21972.635} C_VEL
LIN {X 0,Y 192.756,Z 205.975,A -85,B 0,C 180,E1 -21976.96,E2 -21976.96} C_VEL
LIN {X 0,Y 192.637,Z 205.993,A -85,B 0,C 180,E1 -21981.398,E2 -21981.398} C_VEL
LIN {X 0,Y 192.665,Z 206.016,A -85,B 0,C 180,E1 -21984.227,E2 -21984.227} C_VEL
LIN {X 0,Y 192.86,Z 207.605,A -85,B 0,C 180,E1 -21989.006,E2 -21989.006} C_VEL
LIN {X 0,Y 193.03,Z 209.172,A -85,B 0,C 180,E1 -21993.135,E2 -21993.135} C_VEL
LIN {X 0,Y 193.278,Z 211.296,A -85,B 0,C 180,E1 -21998.183,E2 -21998.183} C_VEL
LIN {X 0,Y 193.487,Z 212.528,A -85,B 0,C 180,E1 -22000.831,E2 -22000.831} C_VEL
LIN {X 0,Y 193.642,Z 213.886,A -85,B 0,C 180,E1 -22003.598,E2 -22003.598} C_VEL
LIN {X 0,Y 193.65,Z 215.413,A -85,B 0,C 180,E1 -22006.541,E2 -22006.541} C_VEL
LIN {X 0,Y 193.306,Z 217.579,A -85,B 0,C 180,E1 -22010.255,E2 -22010.255} C_VEL
LIN {X 0,Y 194.298,Z 220.89,A -85,B 0,C 180,E1 -22010.706,E2 -22010.706} C_VEL
LIN {X 0,Y 195.198,Z 223.168,A -85,B 0,C 180,E1 -22011.102,E2 -22011.102} C_VEL
LIN {X 0,Y 199.068,Z 234.77,A -85,B 0,C 180,E1 -22013.118,E2 -22013.118} C_VEL
LIN {X 0,Y 201.565,Z 244.844,A -85,B 0,C 180,E1 -22014.922,E2 -22014.922} C_VEL
LIN {X 0,Y 203.221,Z 255,A -85,B 0,C 180,E1 -22016.844,E2 -22016.844} C_VEL
LIN {X 0,Y 204.065,Z 263.951,A -85,B 0,C 180,E1 -22018.683,E2 -22018.683} C_VEL
LIN {X 0,Y 204.215,Z 271.867,A -85,B 0,C 180,E1 -22020.445,E2 -22020.445} C_VEL
LIN {X 0,Y 203.903,Z 279.292,A -85,B 0,C 180,E1 -22022.27,E2 -22022.27} C_VEL
LIN {X 0,Y 201.024,Z 288.432,A -85,B 0,C 180,E1 -22024.642,E2 -22024.642} C_VEL
LIN {X 0,Y 198.65,Z 295.534,A -85,B 0,C 180,E1 -22026.906,E2 -22026.906} C_VEL
LIN {X 0,Y 196.764,Z 301.179,A -85,B 0,C 180,E1 -22029.073,E2 -22029.073} C_VEL
LIN {X 0,Y 195.184,Z 305.683,A -85,B 0,C 180,E1 -22031.091,E2 -22031.091} C_VEL
LIN {X 0,Y 193.137,Z 311.176,A -85,B 0,C 180,E1 -22034.162,E2 -22034.162} C_VEL
LIN {X 0,Y 191.733,Z 315.508,A -85,B 0,C 180,E1 -22037.295,E2 -22037.295} C_VEL
LIN {X 0,Y 191.061,Z 317.881,A -85,B 0,C 180,E1 -22039.402,E2 -22039.402} C_VEL
LIN {X 0,Y 190.582,Z 319.685,A -85,B 0,C 180,E1 -22041.518,E2 -22041.518} C_VEL
LIN {X 0,Y 190.167,Z 322.143,A -85,B 0,C 180,E1 -22045.761,E2 -22045.761} C_VEL
LIN {X 0,Y 190.186,Z 322.839,A -85,B 0,C 180,E1 -22049.224,E2 -22049.224} C_VEL
LIN {X 0,Y 190.179,Z 322.739,A -85,B 0,C 180,E1 -22052.118,E2 -22052.118} C_VEL
LIN {X 0,Y 190.168,Z 322.144,A -85,B 0,C 180,E1 -22054.239,E2 -22054.239} C_VEL
LIN {X 0,Y 190.544,Z 319.824,A -85,B 0,C 180,E1 -22058.271,E2 -22058.271} C_VEL
LIN {X 0,Y 190.239,Z 318.501,A -85,B 0,C 180,E1 -22060,E2 -22060} C_VEL
LIN {X 0,Y 188.192,Z 315.66,A -85,B 0,C 180,E1 -22062.811,E2 -22062.811} C_VEL
LIN {X 0,Y 186.692,Z 312.873,A -85,B 0,C 180,E1 -22065.05,E2 -22065.05} C_VEL
LIN {X 0,Y 186.541,Z 310.542,A -85,B 0,C 180,E1 -22066.721,E2 -22066.721} C_VEL
LIN {X 0,Y 186.794,Z 309.673,A -85,B 0,C 180,E1 -22067.266,E2 -22067.266} C_VEL
LIN {X 0,Y 189.202,Z 303.277,A -85,B 0,C 180,E1 -22070.663,E2 -22070.663} C_VEL
LIN {X 0,Y 191.548,Z 297.082,A -85,B 0,C 180,E1 -22073.27,E2 -22073.27} C_VEL
LIN {X 0,Y 193.467,Z 291.474,A -85,B 0,C 180,E1 -22075.267,E2 -22075.267} C_VEL
LIN {X 0,Y 196.405,Z 282.921,A -85,B 0,C 180,E1 -22077.721,E2 -22077.721} C_VEL
LIN {X 0,Y 197.382,Z 279.072,A -85,B 0,C 180,E1 -22078.729,E2 -22078.729} C_VEL
LIN {X 0,Y 197.69,Z 268.333,A -85,B 0,C 180,E1 -22081.435,E2 -22081.435} C_VEL
LIN {X 0,Y 197.144,Z 258.677,A -85,B 0,C 180,E1 -22083.589,E2 -22083.589} C_VEL
LIN {X 0,Y 195.816,Z 248.9,A -85,B 0,C 180,E1 -22085.6,E2 -22085.6} C_VEL
LIN {X 0,Y 193.728,Z 239.082,A -85,B 0,C 180,E1 -22087.504,E2 -22087.504} C_VEL
LIN {X 0,Y 190.575,Z 228.659,A -85,B 0,C 180,E1 -22089.474,E2 -22089.474} C_VEL
LIN {X 0,Y 187.915,Z 221.49,A -85,B 0,C 180,E1 -22090.842,E2 -22090.842} C_VEL
LIN {X 0,Y 186.519,Z 218.224,A -85,B 0,C 180,E1 -22091.437,E2 -22091.437} C_VEL
LIN {X 0,Y 186.396,Z 217.279,A -85,B 0,C 180,E1 -22091.587,E2 -22091.587} C_VEL
LIN {X 0,Y 186.556,Z 215.067,A -85,B 0,C 180,E1 -22095.706,E2 -22095.706} C_VEL
LIN {X 0,Y 186.377,Z 212.99,A -85,B 0,C 180,E1 -22100.129,E2 -22100.129} C_VEL
LIN {X 0,Y 186.032,Z 210.743,A -85,B 0,C 180,E1 -22105.48,E2 -22105.48} C_VEL
LIN {X 0,Y 185.845,Z 208.865,A -85,B 0,C 180,E1 -22110.552,E2 -22110.552} C_VEL
LIN {X 0,Y 185.661,Z 207.277,A -85,B 0,C 180,E1 -22115.392,E2 -22115.392} C_VEL
LIN {X 0,Y 185.597,Z 206.873,A -85,B 0,C 180,E1 -22117.747,E2 -22117.747} C_VEL
LIN {X 0,Y 185.689,Z 206.857,A -85,B 0,C 180,E1 -22122.374,E2 -22122.374} C_VEL
LIN {X 0,Y 185.728,Z 206.85,A -85,B 0,C 180,E1 -22126.876,E2 -22126.876} C_VEL
LIN {X 0,Y 185.981,Z 206.819,A -85,B 0,C 180,E1 -22131.305,E2 -22131.305} C_VEL
LIN {X 0,Y 186.203,Z 206.788,A -85,B 0,C 180,E1 -22137.836,E2 -22137.836} C_VEL
LIN {X 0,Y 186.404,Z 206.746,A -85,B 0,C 180,E1 -22139.999,E2 -22139.999} C_VEL
LIN {X 0,Y 185.915,Z 206.809,A -85,B 0,C 180,E1 -22144.335,E2 -22144.335} C_VEL
LIN {X 0,Y 185.98,Z 206.815,A -85,B 0,C 180,E1 -22148.693,E2 -22148.693} C_VEL
LIN {X 0,Y 185.728,Z 206.849,A -85,B 0,C 180,E1 -22153.122,E2 -22153.122} C_VEL
LIN {X 0,Y 185.687,Z 206.855,A -85,B 0,C 180,E1 -22157.624,E2 -22157.624} C_VEL
LIN {X 0,Y 185.594,Z 206.866,A -85,B 0,C 180,E1 -22162.25,E2 -22162.25} C_VEL
LIN {X 0,Y 185.559,Z 206.871,A -85,B 0,C 180,E1 -22167.031,E2 -22167.031} C_VEL
LIN {X 0,Y 185.576,Z 206.869,A -85,B 0,C 180,E1 -22169.492,E2 -22169.492} C_VEL
LIN {X 0,Y 185.516,Z 206.878,A -85,B 0,C 180,E1 -22174.627,E2 -22174.627} C_VEL
LIN {X 0,Y 185.54,Z 206.873,A -85,B 0,C 180,E1 -22177.303,E2 -22177.303} C_VEL
LIN {X 0,Y 185.487,Z 206.879,A -85,B 0,C 180,E1 -22180.731,E2 -22180.731} C_VEL
LIN {X 0,Y 185.48,Z 206.881,A -85,B 0,C 180,E1 -22186.047,E2 -22186.047} C_VEL
LIN {X 0,Y 185.461,Z 206.883,A -85,B 0,C 180,E1 -22188.033,E2 -22188.033} C_VEL
LIN {X 0,Y 186.459,Z 209.736,A -85,B 0,C 180,E1 -22188.535,E2 -22188.535} C_VEL
LIN {X 0,Y 188.293,Z 212.098,A -85,B 0,C 180,E1 -22189.189,E2 -22189.189} C_VEL
LIN {X 0,Y 193.065,Z 220.395,A -85,B 0,C 180,E1 -22191.189,E2 -22191.189} C_VEL
LIN {X 0,Y 198.404,Z 231.12,A -85,B 0,C 180,E1 -22193.691,E2 -22193.691} C_VEL
LIN {X 0,Y 203.121,Z 243.341,A -85,B 0,C 180,E1 -22196.539,E2 -22196.539} C_VEL
LIN {X 0,Y 205.661,Z 252.281,A -85,B 0,C 180,E1 -22198.682,E2 -22198.682} C_VEL
LIN {X 0,Y 208.519,Z 261.519,A -85,B 0,C 180,E1 -22201.198,E2 -22201.198} C_VEL
LIN {X 0,Y 211.856,Z 269.022,A -85,B 0,C 180,E1 -22203.594,E2 -22203.594} C_VEL
LIN {X 0,Y 216.794,Z 277.098,A -85,B 0,C 180,E1 -22206.589,E2 -22206.589} C_VEL
LIN {X 0,Y 223.028,Z 284.388,A -85,B 0,C 180,E1 -22209.719,E2 -22209.719} C_VEL
LIN {X 0,Y 228.769,Z 289.587,A -85,B 0,C 180,E1 -22212.238,E2 -22212.238} C_VEL
LIN {X 0,Y 236.26,Z 294.961,A -85,B 0,C 180,E1 -22215.181,E2 -22215.181} C_VEL
LIN {X 0,Y 245.167,Z 300.081,A -85,B 0,C 180,E1 -22218.424,E2 -22218.424} C_VEL
LIN {X 0,Y 250.516,Z 302.646,A -85,B 0,C 180,E1 -22220.31,E2 -22220.31} C_VEL
LIN {X 0,Y 255.411,Z 304.801,A -85,B 0,C 180,E1 -22222.128,E2 -22222.128} C_VEL
LIN {X 0,Y 261.229,Z 307.067,A -85,B 0,C 180,E1 -22224.512,E2 -22224.512} C_VEL
LIN {X 0,Y 262.949,Z 307.697,A -85,B 0,C 180,E1 -22225.401,E2 -22225.401} C_VEL
LIN {X 0,Y 265.438,Z 308.627,A -85,B 0,C 180,E1 -22226.965,E2 -22226.965} C_VEL
LIN {X 0,Y 267.642,Z 309.144,A -85,B 0,C 180,E1 -22228.495,E2 -22228.495} C_VEL
LIN {X 0,Y 269.032,Z 309.292,A -85,B 0,C 180,E1 -22230,E2 -22230} C_VEL
LIN {X 0,Y 267.197,Z 309.045,A -85,B 0,C 180,E1 -22231.838,E2 -22231.838} C_VEL
LIN {X 0,Y 265.438,Z 308.626,A -85,B 0,C 180,E1 -22233.035,E2 -22233.035} C_VEL
LIN {X 0,Y 262.941,Z 307.696,A -85,B 0,C 180,E1 -22234.599,E2 -22234.599} C_VEL
LIN {X 0,Y 259.506,Z 306.432,A -85,B 0,C 180,E1 -22236.219,E2 -22236.219} C_VEL
LIN {X 0,Y 255.353,Z 304.76,A -85,B 0,C 180,E1 -22237.91,E2 -22237.91} C_VEL
LIN {X 0,Y 247.805,Z 301.384,A -85,B 0,C 180,E1 -22240.663,E2 -22240.663} C_VEL
LIN {X 0,Y 238.857,Z 296.635,A -85,B 0,C 180,E1 -22243.843,E2 -22243.843} C_VEL
LIN {X 0,Y 231.219,Z 291.48,A -85,B 0,C 180,E1 -22246.777,E2 -22246.777} C_VEL
LIN {X 0,Y 224.083,Z 285.433,A -85,B 0,C 180,E1 -22249.8,E2 -22249.8} C_VEL
LIN {X 0,Y 218,Z 278.702,A -85,B 0,C 180,E1 -22252.759,E2 -22252.759} C_VEL
LIN {X 0,Y 213.046,Z 271.324,A -85,B 0,C 180,E1 -22255.596,E2 -22255.596} C_VEL
LIN {X 0,Y 209.548,Z 264.119,A -85,B 0,C 180,E1 -22258.004,E2 -22258.004} C_VEL
LIN {X 0,Y 206.615,Z 255.842,A -85,B 0,C 180,E1 -22260.393,E2 -22260.393} C_VEL
LIN {X 0,Y 204.25,Z 247.19,A -85,B 0,C 180,E1 -22262.544,E2 -22262.544} C_VEL
LIN {X 0,Y 201.624,Z 239.237,A -85,B 0,C 180,E1 -22264.427,E2 -22264.427} C_VEL
LIN {X 0,Y 197.911,Z 230.082,A -85,B 0,C 180,E1 -22266.544,E2 -22266.544} C_VEL
LIN {X 0,Y 192.677,Z 219.626,A -85,B 0,C 180,E1 -22268.98,E2 -22268.98} C_VEL
LIN {X 0,Y 189.627,Z 214.509,A -85,B 0,C 180,E1 -22270.252,E2 -22270.252} C_VEL
LIN {X 0,Y 187.676,Z 211.16,A -85,B 0,C 180,E1 -22271.052,E2 -22271.052} C_VEL
LIN {X 0,Y 185.996,Z 208.766,A -85,B 0,C 180,E1 -22271.684,E2 -22271.684} C_VEL
LIN {X 0,Y 185.47,Z 206.882,A -85,B 0,C 180,E1 -22271.96,E2 -22271.96} C_VEL
LIN {X 0,Y 185.494,Z 206.88,A -85,B 0,C 180,E1 -22276.043,E2 -22276.043} C_VEL
LIN {X 0,Y 185.49,Z 206.879,A -85,B 0,C 180,E1 -22279.903,E2 -22279.903} C_VEL
LIN {X 0,Y 185.54,Z 206.873,A -85,B 0,C 180,E1 -22282.697,E2 -22282.697} C_VEL
LIN {X 0,Y 185.542,Z 206.873,A -85,B 0,C 180,E1 -22287.976,E2 -22287.976} C_VEL
LIN {X 0,Y 185.579,Z 206.869,A -85,B 0,C 180,E1 -22290.577,E2 -22290.577} C_VEL
LIN {X 0,Y 185.584,Z 206.861,A -85,B 0,C 180,E1 -22295.383,E2 -22295.383} C_VEL
LIN {X 0,Y 185.604,Z 206.856,A -85,B 0,C 180,E1 -22300.076,E2 -22300.076} C_VEL
LIN {X 0,Y 185.692,Z 206.848,A -85,B 0,C 180,E1 -22304.638,E2 -22304.638} C_VEL
LIN {X 0,Y 185.886,Z 206.825,A -85,B 0,C 180,E1 -22309.419,E2 -22309.419} C_VEL
LIN {X 0,Y 185.945,Z 206.822,A -85,B 0,C 180,E1 -22313.491,E2 -22313.491} C_VEL
LIN {X 0,Y 186.203,Z 206.757,A -85,B 0,C 180,E1 -22317.838,E2 -22317.838} C_VEL
LIN {X 0,Y 186.404,Z 206.746,A -85,B 0,C 180,E1 -22320.001,E2 -22320.001} C_VEL
LIN {X 0,Y 185.916,Z 206.826,A -85,B 0,C 180,E1 -22324.337,E2 -22324.337} C_VEL
LIN {X 0,Y 185.981,Z 206.819,A -85,B 0,C 180,E1 -22328.695,E2 -22328.695} C_VEL
LIN {X 0,Y 185.728,Z 206.851,A -85,B 0,C 180,E1 -22333.124,E2 -22333.124} C_VEL
LIN {X 0,Y 185.689,Z 206.856,A -85,B 0,C 180,E1 -22337.626,E2 -22337.626} C_VEL
LIN {X 0,Y 185.597,Z 206.866,A -85,B 0,C 180,E1 -22342.253,E2 -22342.253} C_VEL
LIN {X 0,Y 185.651,Z 207.302,A -85,B 0,C 180,E1 -22344.697,E2 -22344.697} C_VEL
LIN {X 0,Y 185.852,Z 208.905,A -85,B 0,C 180,E1 -22349.573,E2 -22349.573} C_VEL
LIN {X 0,Y 186.034,Z 210.742,A -85,B 0,C 180,E1 -22354.52,E2 -22354.52} C_VEL
LIN {X 0,Y 186.382,Z 212.997,A -85,B 0,C 180,E1 -22359.87,E2 -22359.87} C_VEL
LIN {X 0,Y 186.557,Z 215.09,A -85,B 0,C 180,E1 -22364.295,E2 -22364.295} C_VEL
LIN {X 0,Y 186.398,Z 217.264,A -85,B 0,C 180,E1 -22368.412,E2 -22368.412} C_VEL
LIN {X 0,Y 187.378,Z 220.542,A -85,B 0,C 180,E1 -22368.946,E2 -22368.946} C_VEL
LIN {X 0,Y 188.47,Z 222.673,A -85,B 0,C 180,E1 -22369.409,E2 -22369.409} C_VEL
LIN {X 0,Y 192.213,Z 233.551,A -85,B 0,C 180,E1 -22371.445,E2 -22371.445} C_VEL
LIN {X 0,Y 194.984,Z 244.513,A -85,B 0,C 180,E1 -22373.538,E2 -22373.538} C_VEL
LIN {X 0,Y 196.553,Z 253.498,A -85,B 0,C 180,E1 -22375.327,E2 -22375.327} C_VEL
LIN {X 0,Y 197.495,Z 263.009,A -85,B 0,C 180,E1 -22377.359,E2 -22377.359} C_VEL
LIN {X 0,Y 197.687,Z 272.202,A -85,B 0,C 180,E1 -22379.511,E2 -22379.511} C_VEL
LIN {X 0,Y 197.382,Z 279.072,A -85,B 0,C 180,E1 -22381.271,E2 -22381.271} C_VEL
LIN {X 0,Y 195.796,Z 284.84,A -85,B 0,C 180,E1 -22382.765,E2 -22382.765} C_VEL
LIN {X 0,Y 192.442,Z 294.424,A -85,B 0,C 180,E1 -22385.742,E2 -22385.742} C_VEL
LIN {X 0,Y 190.146,Z 300.968,A -85,B 0,C 180,E1 -22388.309,E2 -22388.309} C_VEL
LIN {X 0,Y 188.443,Z 305.471,A -85,B 0,C 180,E1 -22390.388,E2 -22390.388} C_VEL
LIN {X 0,Y 186.286,Z 310.964,A -85,B 0,C 180,E1 -22393.564,E2 -22393.564} C_VEL
LIN {X 0,Y 184.792,Z 315.296,A -85,B 0,C 180,E1 -22396.81,E2 -22396.81} C_VEL
LIN {X 0,Y 184.069,Z 317.669,A -85,B 0,C 180,E1 -22398.994,E2 -22398.994} C_VEL
LIN {X 0,Y 183.546,Z 319.473,A -85,B 0,C 180,E1 -22401.19,E2 -22401.19} C_VEL
LIN {X 0,Y 183.081,Z 321.932,A -85,B 0,C 180,E1 -22405.597,E2 -22405.597} C_VEL
LIN {X 0,Y 183.076,Z 322.527,A -85,B 0,C 180,E1 -22407.8,E2 -22407.8} C_VEL
LIN {X 0,Y 183.145,Z 322.685,A -85,B 0,C 180,E1 -22410,E2 -22410} C_VEL
LIN {X 0,Y 183.056,Z 322.199,A -85,B 0,C 180,E1 -22413.414,E2 -22413.414} C_VEL
LIN {X 0,Y 183.231,Z 320.867,A -85,B 0,C 180,E1 -22416.607,E2 -22416.607} C_VEL
LIN {X 0,Y 183.547,Z 319.473,A -85,B 0,C 180,E1 -22418.81,E2 -22418.81} C_VEL
LIN {X 0,Y 184.389,Z 316.516,A -85,B 0,C 180,E1 -22422.101,E2 -22422.101} C_VEL
LIN {X 0,Y 185.679,Z 312.519,A -85,B 0,C 180,E1 -22425.364,E2 -22425.364} C_VEL
LIN {X 0,Y 186.794,Z 309.673,A -85,B 0,C 180,E1 -22427.266,E2 -22427.266} C_VEL
LIN {X 0,Y 187.199,Z 307.027,A -85,B 0,C 180,E1 -22428.881,E2 -22428.881} C_VEL
LIN {X 0,Y 186.268,Z 302.195,A -85,B 0,C 180,E1 -22431.528,E2 -22431.528} C_VEL
LIN {X 0,Y 185.577,Z 296.85,A -85,B 0,C 180,E1 -22434.095,E2 -22434.095} C_VEL
LIN {X 0,Y 186.347,Z 293.215,A -85,B 0,C 180,E1 -22435.536,E2 -22435.536} C_VEL
LIN {X 0,Y 189.465,Z 284.627,A -85,B 0,C 180,E1 -22438.225,E2 -22438.225} C_VEL
LIN {X 0,Y 190.645,Z 280.784,A -85,B 0,C 180,E1 -22439.238,E2 -22439.238} C_VEL
LIN {X 0,Y 191.185,Z 273.128,A -85,B 0,C 180,E1 -22441.333,E2 -22441.333} C_VEL
LIN {X 0,Y 191.175,Z 265.741,A -85,B 0,C 180,E1 -22443.179,E2 -22443.179} C_VEL
LIN {X 0,Y 190.545,Z 257.218,A -85,B 0,C 180,E1 -22445.156,E2 -22445.156} C_VEL
LIN {X 0,Y 189.256,Z 248.072,A -85,B 0,C 180,E1 -22447.132,E2 -22447.132} C_VEL
LIN {X 0,Y 187.011,Z 238.196,A -85,B 0,C 180,E1 -22449.185,E2 -22449.185} C_VEL
LIN {X 0,Y 183.922,Z 228.294,A -85,B 0,C 180,E1 -22451.214,E2 -22451.214} C_VEL
LIN {X 0,Y 181.145,Z 221.435,A -85,B 0,C 180,E1 -22452.701,E2 -22452.701} C_VEL
LIN {X 0,Y 179.705,Z 218.28,A -85,B 0,C 180,E1 -22453.361,E2 -22453.361} C_VEL
LIN {X 0,Y 179.479,Z 217.014,A -85,B 0,C 180,E1 -22453.569,E2 -22453.569} C_VEL
LIN {X 0,Y 179.408,Z 214.745,A -85,B 0,C 180,E1 -22458.244,E2 -22458.244} C_VEL
LIN {X 0,Y 179.204,Z 213.278,A -85,B 0,C 180,E1 -22461.66,E2 -22461.66} C_VEL
LIN {X 0,Y 178.944,Z 211.295,A -85,B 0,C 180,E1 -22466.642,E2 -22466.642} C_VEL
LIN {X 0,Y 178.728,Z 209.496,A -85,B 0,C 180,E1 -22471.843,E2 -22471.843} C_VEL
LIN {X 0,Y 178.55,Z 207.988,A -85,B 0,C 180,E1 -22476.819,E2 -22476.819} C_VEL
LIN {X 0,Y 178.649,Z 207.735,A -85,B 0,C 180,E1 -22481.655,E2 -22481.655} C_VEL
LIN {X 0,Y 178.656,Z 207.732,A -85,B 0,C 180,E1 -22486.346,E2 -22486.346} C_VEL
LIN {X 0,Y 178.91,Z 207.699,A -85,B 0,C 180,E1 -22490.958,E2 -22490.958} C_VEL
LIN {X 0,Y 179.149,Z 207.667,A -85,B 0,C 180,E1 -22497.75,E2 -22497.75} C_VEL
LIN {X 0,Y 179.367,Z 207.621,A -85,B 0,C 180,E1 -22499.999,E2 -22499.999} C_VEL
LIN {X 0,Y 178.862,Z 207.688,A -85,B 0,C 180,E1 -22504.506,E2 -22504.506} C_VEL
LIN {X 0,Y 178.909,Z 207.693,A -85,B 0,C 180,E1 -22509.039,E2 -22509.039} C_VEL
LIN {X 0,Y 178.656,Z 207.727,A -85,B 0,C 180,E1 -22513.651,E2 -22513.651} C_VEL
LIN {X 0,Y 178.62,Z 207.728,A -85,B 0,C 180,E1 -22519.215,E2 -22519.215} C_VEL
LIN {X 0,Y 178.521,Z 207.74,A -85,B 0,C 180,E1 -22525.117,E2 -22525.117} C_VEL
LIN {X 0,Y 178.52,Z 207.748,A -85,B 0,C 180,E1 -22529.993,E2 -22529.993} C_VEL
LIN {X 0,Y 178.492,Z 207.75,A -85,B 0,C 180,E1 -22534.224,E2 -22534.224} C_VEL
LIN {X 0,Y 178.417,Z 207.762,A -85,B 0,C 180,E1 -22539.067,E2 -22539.067} C_VEL
LIN {X 0,Y 178.413,Z 207.762,A -85,B 0,C 180,E1 -22542.039,E2 -22542.039} C_VEL
LIN {X 0,Y 178.449,Z 207.765,A -85,B 0,C 180,E1 -22546.051,E2 -22546.051} C_VEL
LIN {X 0,Y 179.423,Z 210.598,A -85,B 0,C 180,E1 -22546.56,E2 -22546.56} C_VEL
LIN {X 0,Y 181.374,Z 213.069,A -85,B 0,C 180,E1 -22547.327,E2 -22547.327} C_VEL
LIN {X 0,Y 183.319,Z 216.338,A -85,B 0,C 180,E1 -22548.225,E2 -22548.225} C_VEL
LIN {X 0,Y 187.791,Z 224.096,A -85,B 0,C 180,E1 -22550.269,E2 -22550.269} C_VEL
LIN {X 0,Y 192.696,Z 234.535,A -85,B 0,C 180,E1 -22552.914,E2 -22552.914} C_VEL
LIN {X 0,Y 196.405,Z 244.354,A -85,B 0,C 180,E1 -22555.386,E2 -22555.386} C_VEL
LIN {X 0,Y 198.723,Z 252.068,A -85,B 0,C 180,E1 -22557.356,E2 -22557.356} C_VEL
LIN {X 0,Y 201.145,Z 261.421,A -85,B 0,C 180,E1 -22559.949,E2 -22559.949} C_VEL
LIN {X 0,Y 204.05,Z 269.212,A -85,B 0,C 180,E1 -22562.482,E2 -22562.482} C_VEL
LIN {X 0,Y 208.435,Z 277.26,A -85,B 0,C 180,E1 -22565.556,E2 -22565.556} C_VEL
LIN {X 0,Y 213.129,Z 283.482,A -85,B 0,C 180,E1 -22568.276,E2 -22568.276} C_VEL
LIN {X 0,Y 219.237,Z 289.564,A -85,B 0,C 180,E1 -22571.303,E2 -22571.303} C_VEL
LIN {X 0,Y 226.274,Z 294.894,A -85,B 0,C 180,E1 -22574.329,E2 -22574.329} C_VEL
LIN {X 0,Y 233.55,Z 299.245,A -85,B 0,C 180,E1 -22577.151,E2 -22577.151} C_VEL
LIN {X 0,Y 242.389,Z 303.383,A -85,B 0,C 180,E1 -22580.333,E2 -22580.333} C_VEL
LIN {X 0,Y 248.128,Z 305.663,A -85,B 0,C 180,E1 -22582.448,E2 -22582.448} C_VEL
LIN {X 0,Y 254.037,Z 307.651,A -85,B 0,C 180,E1 -22584.829,E2 -22584.829} C_VEL
LIN {X 0,Y 257.781,Z 308.857,A -85,B 0,C 180,E1 -22586.874,E2 -22586.874} C_VEL
LIN {X 0,Y 260.168,Z 309.366,A -85,B 0,C 180,E1 -22588.452,E2 -22588.452} C_VEL
LIN {X 0,Y 261.781,Z 309.504,A -85,B 0,C 180,E1 -22590,E2 -22590} C_VEL
LIN {X 0,Y 260.131,Z 309.354,A -85,B 0,C 180,E1 -22591.587,E2 -22591.587} C_VEL
LIN {X 0,Y 257.778,Z 308.856,A -85,B 0,C 180,E1 -22593.126,E2 -22593.126} C_VEL
LIN {X 0,Y 254.037,Z 307.652,A -85,B 0,C 180,E1 -22595.17,E2 -22595.17} C_VEL
LIN {X 0,Y 248.134,Z 305.649,A -85,B 0,C 180,E1 -22597.563,E2 -22597.563} C_VEL
LIN {X 0,Y 241.27,Z 302.92,A -85,B 0,C 180,E1 -22600.065,E2 -22600.065} C_VEL
LIN {X 0,Y 231.42,Z 298.125,A -85,B 0,C 180,E1 -22603.642,E2 -22603.642} C_VEL
LIN {X 0,Y 223.722,Z 293.122,A -85,B 0,C 180,E1 -22606.742,E2 -22606.742} C_VEL
LIN {X 0,Y 216.741,Z 287.282,A -85,B 0,C 180,E1 -22609.893,E2 -22609.893} C_VEL
LIN {X 0,Y 210.402,Z 280.149,A -85,B 0,C 180,E1 -22613.236,E2 -22613.236} C_VEL
LIN {X 0,Y 205.526,Z 272.295,A -85,B 0,C 180,E1 -22616.393,E2 -22616.393} C_VEL
LIN {X 0,Y 202.518,Z 265.357,A -85,B 0,C 180,E1 -22618.811,E2 -22618.811} C_VEL
LIN {X 0,Y 200.08,Z 257.801,A -85,B 0,C 180,E1 -22621.112,E2 -22621.112} C_VEL
LIN {X 0,Y 197.79,Z 248.727,A -85,B 0,C 180,E1 -22623.497,E2 -22623.497} C_VEL
LIN {X 0,Y 194.392,Z 238.818,A -85,B 0,C 180,E1 -22626.008,E2 -22626.008} C_VEL
LIN {X 0,Y 190.876,Z 230.522,A -85,B 0,C 180,E1 -22628.101,E2 -22628.101} C_VEL
LIN {X 0,Y 185.709,Z 220.326,A -85,B 0,C 180,E1 -22630.698,E2 -22630.698} C_VEL
LIN {X 0,Y 182.782,Z 215.66,A -85,B 0,C 180,E1 -22632,E2 -22632} C_VEL
LIN {X 0,Y 180.74,Z 212.124,A -85,B 0,C 180,E1 -22632.939,E2 -22632.939} C_VEL
LIN {X 0,Y 179.04,Z 209.814,A -85,B 0,C 180,E1 -22633.638,E2 -22633.638} C_VEL
LIN {X 0,Y 178.483,Z 207.753,A -85,B 0,C 180,E1 -22634.011,E2 -22634.011} C_VEL
LIN {X 0,Y 178.417,Z 207.761,A -85,B 0,C 180,E1 -22638.453,E2 -22638.453} C_VEL
LIN {X 0,Y 178.446,Z 207.756,A -85,B 0,C 180,E1 -22643.79,E2 -22643.79} C_VEL
LIN {X 0,Y 178.487,Z 207.75,A -85,B 0,C 180,E1 -22646.548,E2 -22646.548} C_VEL
LIN {X 0,Y 178.52,Z 207.748,A -85,B 0,C 180,E1 -22650.007,E2 -22650.007} C_VEL
LIN {X 0,Y 178.521,Z 207.74,A -85,B 0,C 180,E1 -22654.883,E2 -22654.883} C_VEL
LIN {X 0,Y 178.62,Z 207.728,A -85,B 0,C 180,E1 -22660.785,E2 -22660.785} C_VEL
LIN {X 0,Y 178.656,Z 207.727,A -85,B 0,C 180,E1 -22666.349,E2 -22666.349} C_VEL
LIN {X 0,Y 178.909,Z 207.693,A -85,B 0,C 180,E1 -22670.961,E2 -22670.961} C_VEL
LIN {X 0,Y 178.862,Z 207.688,A -85,B 0,C 180,E1 -22675.494,E2 -22675.494} C_VEL
LIN {X 0,Y 179.367,Z 207.621,A -85,B 0,C 180,E1 -22680.001,E2 -22680.001} C_VEL
LIN {X 0,Y 178.864,Z 207.705,A -85,B 0,C 180,E1 -22684.508,E2 -22684.508} C_VEL
LIN {X 0,Y 178.91,Z 207.7,A -85,B 0,C 180,E1 -22689.042,E2 -22689.042} C_VEL
LIN {X 0,Y 178.656,Z 207.733,A -85,B 0,C 180,E1 -22693.654,E2 -22693.654} C_VEL
LIN {X 0,Y 178.623,Z 207.735,A -85,B 0,C 180,E1 -22699.217,E2 -22699.217} C_VEL
LIN {X 0,Y 178.55,Z 207.979,A -85,B 0,C 180,E1 -22703.181,E2 -22703.181} C_VEL
LIN {X 0,Y 178.728,Z 209.492,A -85,B 0,C 180,E1 -22708.157,E2 -22708.157} C_VEL
LIN {X 0,Y 178.851,Z 210.346,A -85,B 0,C 180,E1 -22710.721,E2 -22710.721} C_VEL
LIN {X 0,Y 179.044,Z 212.361,A -85,B 0,C 180,E1 -22716.073,E2 -22716.073} C_VEL
LIN {X 0,Y 179.241,Z 213.496,A -85,B 0,C 180,E1 -22718.857,E2 -22718.857} C_VEL
LIN {X 0,Y 179.411,Z 214.821,A -85,B 0,C 180,E1 -22721.904,E2 -22721.904} C_VEL
LIN {X 0,Y 179.463,Z 217.032,A -85,B 0,C 180,E1 -22726.437,E2 -22726.437} C_VEL
LIN {X 0,Y 180.526,Z 220.36,A -85,B 0,C 180,E1 -22727.031,E2 -22727.031} C_VEL
LIN {X 0,Y 181.739,Z 222.666,A -85,B 0,C 180,E1 -22727.593,E2 -22727.593} C_VEL
LIN {X 0,Y 184.745,Z 230.417,A -85,B 0,C 180,E1 -22729.224,E2 -22729.224} C_VEL
LIN {X 0,Y 188.125,Z 242.46,A -85,B 0,C 180,E1 -22731.678,E2 -22731.678} C_VEL
LIN {X 0,Y 190.093,Z 253.543,A -85,B 0,C 180,E1 -22734.024,E2 -22734.024} C_VEL
LIN {X 0,Y 191.027,Z 263.081,A -85,B 0,C 180,E1 -22736.177,E2 -22736.177} C_VEL
LIN {X 0,Y 191.233,Z 271.773,A -85,B 0,C 180,E1 -22738.31,E2 -22738.31} C_VEL
LIN {X 0,Y 190.879,Z 278.85,A -85,B 0,C 180,E1 -22740.195,E2 -22740.195} C_VEL
LIN {X 0,Y 190.131,Z 282.709,A -85,B 0,C 180,E1 -22741.28,E2 -22741.28} C_VEL
LIN {X 0,Y 187.033,Z 291.262,A -85,B 0,C 180,E1 -22743.8,E2 -22743.8} C_VEL
LIN {X 0,Y 184.18,Z 299.304,A -85,B 0,C 180,E1 -22746.826,E2 -22746.826} C_VEL
LIN {X 0,Y 181.722,Z 305.258,A -85,B 0,C 180,E1 -22749.631,E2 -22749.631} C_VEL
LIN {X 0,Y 179.46,Z 310.752,A -85,B 0,C 180,E1 -22752.92,E2 -22752.92} C_VEL
LIN {X 0,Y 177.847,Z 315.084,A -85,B 0,C 180,E1 -22756.285,E2 -22756.285} C_VEL
LIN {X 0,Y 177.066,Z 317.456,A -85,B 0,C 180,E1 -22758.553,E2 -22758.553} C_VEL
LIN {X 0,Y 176.504,Z 319.261,A -85,B 0,C 180,E1 -22760.836,E2 -22760.836} C_VEL
LIN {X 0,Y 176.011,Z 321.721,A -85,B 0,C 180,E1 -22765.42,E2 -22765.42} C_VEL
LIN {X 0,Y 175.975,Z 322.315,A -85,B 0,C 180,E1 -22767.711,E2 -22767.711} C_VEL
LIN {X 0,Y 176.054,Z 322.474,A -85,B 0,C 180,E1 -22770,E2 -22770} C_VEL
LIN {X 0,Y 175.956,Z 322.112,A -85,B 0,C 180,E1 -22773.074,E2 -22773.074} C_VEL
LIN {X 0,Y 176.157,Z 320.655,A -85,B 0,C 180,E1 -22776.874,E2 -22776.874} C_VEL
LIN {X 0,Y 176.505,Z 319.261,A -85,B 0,C 180,E1 -22779.164,E2 -22779.164} C_VEL
LIN {X 0,Y 177.438,Z 316.304,A -85,B 0,C 180,E1 -22782.582,E2 -22782.582} C_VEL
LIN {X 0,Y 178.807,Z 312.306,A -85,B 0,C 180,E1 -22785.97,E2 -22785.97} C_VEL
LIN {X 0,Y 180.931,Z 307.175,A -85,B 0,C 180,E1 -22789.279,E2 -22789.279} C_VEL
LIN {X 0,Y 183.054,Z 301.911,A -85,B 0,C 180,E1 -22791.983,E2 -22791.983} C_VEL
LIN {X 0,Y 184.787,Z 297.496,A -85,B 0,C 180,E1 -22793.903,E2 -22793.903} C_VEL
LIN {X 0,Y 186.347,Z 293.215,A -85,B 0,C 180,E1 -22795.536,E2 -22795.536} C_VEL
LIN {X 0,Y 187.117,Z 289.483,A -85,B 0,C 180,E1 -22796.926,E2 -22796.926} C_VEL
LIN {X 0,Y 186.868,Z 285.669,A -85,B 0,C 180,E1 -22798.328,E2 -22798.328} C_VEL
LIN {X 0,Y 185.223,Z 277.789,A -85,B 0,C 180,E1 -22801.09,E2 -22801.09} C_VEL
LIN {X 0,Y 184.797,Z 271.908,A -85,B 0,C 180,E1 -22802.828,E2 -22802.828} C_VEL
LIN {X 0,Y 184.668,Z 263.153,A -85,B 0,C 180,E1 -22805.081,E2 -22805.081} C_VEL
LIN {X 0,Y 183.713,Z 253.198,A -85,B 0,C 180,E1 -22807.456,E2 -22807.456} C_VEL
LIN {X 0,Y 181.503,Z 241.481,A -85,B 0,C 180,E1 -22810.115,E2 -22810.115} C_VEL
LIN {X 0,Y 178.19,Z 230.14,A -85,B 0,C 180,E1 -22812.622,E2 -22812.622} C_VEL
LIN {X 0,Y 175.759,Z 224.629,A -85,B 0,C 180,E1 -22813.964,E2 -22813.964} C_VEL
LIN {X 0,Y 174.476,Z 221.519,A -85,B 0,C 180,E1 -22814.72,E2 -22814.72} C_VEL
LIN {X 0,Y 172.856,Z 218.623,A -85,B 0,C 180,E1 -22815.496,E2 -22815.496} C_VEL
LIN {X 0,Y 172.398,Z 216.72,A -85,B 0,C 180,E1 -22815.869,E2 -22815.869} C_VEL
LIN {X 0,Y 172.205,Z 214.564,A -85,B 0,C 180,E1 -22820.842,E2 -22820.842} C_VEL
LIN {X 0,Y 171.99,Z 212.896,A -85,B 0,C 180,E1 -22825.103,E2 -22825.103} C_VEL
LIN {X 0,Y 171.735,Z 210.954,A -85,B 0,C 180,E1 -22830.587,E2 -22830.587} C_VEL
LIN {X 0,Y 171.559,Z 209.384,A -85,B 0,C 180,E1 -22835.815,E2 -22835.815} C_VEL
LIN {X 0,Y 171.475,Z 208.706,A -85,B 0,C 180,E1 -22838.353,E2 -22838.353} C_VEL
LIN {X 0,Y 171.579,Z 208.616,A -85,B 0,C 180,E1 -22840.87,E2 -22840.87} C_VEL
LIN {X 0,Y 171.574,Z 208.614,A -85,B 0,C 180,E1 -22845.771,E2 -22845.771} C_VEL
LIN {X 0,Y 171.846,Z 208.58,A -85,B 0,C 180,E1 -22850.584,E2 -22850.584} C_VEL
LIN {X 0,Y 171.812,Z 208.584,A -85,B 0,C 180,E1 -22855.306,E2 -22855.306} C_VEL
LIN {X 0,Y 172.33,Z 208.495,A -85,B 0,C 180,E1 -22859.999,E2 -22859.999} C_VEL
LIN {X 0,Y 171.81,Z 208.567,A -85,B 0,C 180,E1 -22864.691,E2 -22864.691} C_VEL
LIN {X 0,Y 171.845,Z 208.571,A -85,B 0,C 180,E1 -22869.414,E2 -22869.414} C_VEL
LIN {X 0,Y 171.573,Z 208.607,A -85,B 0,C 180,E1 -22874.226,E2 -22874.226} C_VEL
LIN {X 0,Y 171.541,Z 208.608,A -85,B 0,C 180,E1 -22879.561,E2 -22879.561} C_VEL
LIN {X 0,Y 171.459,Z 208.62,A -85,B 0,C 180,E1 -22885.611,E2 -22885.611} C_VEL
LIN {X 0,Y 171.438,Z 208.63,A -85,B 0,C 180,E1 -22890.586,E2 -22890.586} C_VEL
LIN {X 0,Y 171.403,Z 208.634,A -85,B 0,C 180,E1 -22895.031,E2 -22895.031} C_VEL
LIN {X 0,Y 171.378,Z 208.637,A -85,B 0,C 180,E1 -22898.817,E2 -22898.817} C_VEL
LIN {X 0,Y 171.338,Z 208.793,A -85,B 0,C 180,E1 -22903.771,E2 -22903.771} C_VEL
LIN {X 0,Y 172.33,Z 211.453,A -85,B 0,C 180,E1 -22904.327,E2 -22904.327} C_VEL
LIN {X 0,Y 174.431,Z 213.97,A -85,B 0,C 180,E1 -22905.247,E2 -22905.247} C_VEL
LIN {X 0,Y 176.353,Z 217.266,A -85,B 0,C 180,E1 -22906.244,E2 -22906.244} C_VEL
LIN {X 0,Y 180.872,Z 224.877,A -85,B 0,C 180,E1 -22908.497,E2 -22908.497} C_VEL
LIN {X 0,Y 185.64,Z 234.753,A -85,B 0,C 180,E1 -22911.241,E2 -22911.241} C_VEL
LIN {X 0,Y 189.356,Z 244.241,A -85,B 0,C 180,E1 -22913.827,E2 -22913.827} C_VEL
LIN {X 0,Y 192.039,Z 252.995,A -85,B 0,C 180,E1 -22916.235,E2 -22916.235} C_VEL
LIN {X 0,Y 194.092,Z 261.714,A -85,B 0,C 180,E1 -22918.752,E2 -22918.752} C_VEL
LIN {X 0,Y 196.344,Z 268.966,A -85,B 0,C 180,E1 -22921.149,E2 -22921.149} C_VEL
LIN {X 0,Y 199.571,Z 276.114,A -85,B 0,C 180,E1 -22923.893,E2 -22923.893} C_VEL
LIN {X 0,Y 204.547,Z 283.78,A -85,B 0,C 180,E1 -22927.327,E2 -22927.327} C_VEL
LIN {X 0,Y 210.233,Z 289.842,A -85,B 0,C 180,E1 -22930.471,E2 -22930.471} C_VEL
LIN {X 0,Y 216.617,Z 294.961,A -85,B 0,C 180,E1 -22933.494,E2 -22933.494} C_VEL
LIN {X 0,Y 224,Z 299.474,A -85,B 0,C 180,E1 -22936.558,E2 -22936.558} C_VEL
LIN {X 0,Y 231.794,Z 303.201,A -85,B 0,C 180,E1 -22939.519,E2 -22939.519} C_VEL
LIN {X 0,Y 237.282,Z 305.305,A -85,B 0,C 180,E1 -22941.484,E2 -22941.484} C_VEL
LIN {X 0,Y 242.26,Z 306.951,A -85,B 0,C 180,E1 -22943.336,E2 -22943.336} C_VEL
LIN {X 0,Y 246.843,Z 308.24,A -85,B 0,C 180,E1 -22945.195,E2 -22945.195} C_VEL
LIN {X 0,Y 250.009,Z 309.09,A -85,B 0,C 180,E1 -22946.777,E2 -22946.777} C_VEL
LIN {X 0,Y 253.068,Z 309.659,A -85,B 0,C 180,E1 -22948.702,E2 -22948.702} C_VEL
LIN {X 0,Y 254.48,Z 309.717,A -85,B 0,C 180,E1 -22950,E2 -22950} C_VEL
LIN {X 0,Y 252.621,Z 309.589,A -85,B 0,C 180,E1 -22951.594,E2 -22951.594} C_VEL
LIN {X 0,Y 250.004,Z 309.09,A -85,B 0,C 180,E1 -22953.223,E2 -22953.223} C_VEL
LIN {X 0,Y 246.596,Z 308.179,A -85,B 0,C 180,E1 -22954.905,E2 -22954.905} C_VEL
LIN {X 0,Y 240.852,Z 306.476,A -85,B 0,C 180,E1 -22957.21,E2 -22957.21} C_VEL
LIN {X 0,Y 235.028,Z 304.467,A -85,B 0,C 180,E1 -22959.328,E2 -22959.328} C_VEL
LIN {X 0,Y 226.207,Z 300.652,A -85,B 0,C 180,E1 -22962.561,E2 -22962.561} C_VEL
LIN {X 0,Y 218.842,Z 296.436,A -85,B 0,C 180,E1 -22965.546,E2 -22965.546} C_VEL
LIN {X 0,Y 211.619,Z 291.066,A -85,B 0,C 180,E1 -22968.833,E2 -22968.833} C_VEL
LIN {X 0,Y 205.499,Z 284.933,A -85,B 0,C 180,E1 -22972.098,E2 -22972.098} C_VEL
LIN {X 0,Y 201.299,Z 279.118,A -85,B 0,C 180,E1 -22974.807,E2 -22974.807} C_VEL
LIN {X 0,Y 197.772,Z 272.546,A -85,B 0,C 180,E1 -22977.514,E2 -22977.514} C_VEL
LIN {X 0,Y 194.871,Z 264.602,A -85,B 0,C 180,E1 -22980.325,E2 -22980.325} C_VEL
LIN {X 0,Y 193.059,Z 257.249,A -85,B 0,C 180,E1 -22982.561,E2 -22982.561} C_VEL
LIN {X 0,Y 191.323,Z 250.297,A -85,B 0,C 180,E1 -22984.521,E2 -22984.521} C_VEL
LIN {X 0,Y 187.96,Z 240.44,A -85,B 0,C 180,E1 -22987.211,E2 -22987.211} C_VEL
LIN {X 0,Y 184.337,Z 231.884,A -85,B 0,C 180,E1 -22989.558,E2 -22989.558} C_VEL
LIN {X 0,Y 178.839,Z 221.321,A -85,B 0,C 180,E1 -22992.539,E2 -22992.539} C_VEL
LIN {X 0,Y 176.1,Z 216.913,A -85,B 0,C 180,E1 -22993.877,E2 -22993.877} C_VEL
LIN {X 0,Y 173.938,Z 213.253,A -85,B 0,C 180,E1 -22994.985,E2 -22994.985} C_VEL
LIN {X 0,Y 172.031,Z 210.925,A -85,B 0,C 180,E1 -22995.837,E2 -22995.837} C_VEL
LIN {X 0,Y 171.353,Z 208.641,A -85,B 0,C 180,E1 -22996.296,E2 -22996.296} C_VEL
LIN {X 0,Y 171.411,Z 208.632,A -85,B 0,C 180,E1 -23002.049,E2 -23002.049} C_VEL
LIN {X 0,Y 171.407,Z 208.634,A -85,B 0,C 180,E1 -23005.087,E2 -23005.087} C_VEL
LIN {X 0,Y 171.446,Z 208.629,A -85,B 0,C 180,E1 -23010.535,E2 -23010.535} C_VEL
LIN {X 0,Y 171.45,Z 208.622,A -85,B 0,C 180,E1 -23015.802,E2 -23015.802} C_VEL
LIN {X 0,Y 171.576,Z 208.606,A -85,B 0,C 180,E1 -23020.873,E2 -23020.873} C_VEL
LIN {X 0,Y 171.573,Z 208.607,A -85,B 0,C 180,E1 -23025.774,E2 -23025.774} C_VEL
LIN {X 0,Y 171.845,Z 208.571,A -85,B 0,C 180,E1 -23030.586,E2 -23030.586} C_VEL
LIN {X 0,Y 171.81,Z 208.567,A -85,B 0,C 180,E1 -23035.309,E2 -23035.309} C_VEL
LIN {X 0,Y 172.33,Z 208.495,A -85,B 0,C 180,E1 -23040.001,E2 -23040.001} C_VEL
LIN {X 0,Y 171.812,Z 208.583,A -85,B 0,C 180,E1 -23044.694,E2 -23044.694} C_VEL
LIN {X 0,Y 171.846,Z 208.58,A -85,B 0,C 180,E1 -23049.416,E2 -23049.416} C_VEL
LIN {X 0,Y 171.574,Z 208.614,A -85,B 0,C 180,E1 -23054.229,E2 -23054.229} C_VEL
LIN {X 0,Y 171.544,Z 208.617,A -85,B 0,C 180,E1 -23059.563,E2 -23059.563} C_VEL
LIN {X 0,Y 171.475,Z 208.7,A -85,B 0,C 180,E1 -23061.647,E2 -23061.647} C_VEL
LIN {X 0,Y 171.628,Z 210.13,A -85,B 0,C 180,E1 -23066.773,E2 -23066.773} C_VEL
LIN {X 0,Y 171.827,Z 211.429,A -85,B 0,C 180,E1 -23070.805,E2 -23070.805} C_VEL
LIN {X 0,Y 171.996,Z 213.015,A -85,B 0,C 180,E1 -23075.193,E2 -23075.193} C_VEL
LIN {X 0,Y 172.208,Z 214.567,A -85,B 0,C 180,E1 -23079.159,E2 -23079.159} C_VEL
LIN {X 0,Y 172.405,Z 216.791,A -85,B 0,C 180,E1 -23084.194,E2 -23084.194} C_VEL
LIN {X 0,Y 173.492,Z 219.969,A -85,B 0,C 180,E1 -23084.819,E2 -23084.819} C_VEL
LIN {X 0,Y 174.989,Z 222.504,A -85,B 0,C 180,E1 -23085.553,E2 -23085.553} C_VEL
LIN {X 0,Y 178.506,Z 231.104,A -85,B 0,C 180,E1 -23087.581,E2 -23087.581} C_VEL
LIN {X 0,Y 181.947,Z 243.434,A -85,B 0,C 180,E1 -23090.338,E2 -23090.338} C_VEL
LIN {X 0,Y 183.714,Z 253.196,A -85,B 0,C 180,E1 -23092.543,E2 -23092.543} C_VEL
LIN {X 0,Y 184.668,Z 263.151,A -85,B 0,C 180,E1 -23094.918,E2 -23094.918} C_VEL
LIN {X 0,Y 184.838,Z 271.548,A -85,B 0,C 180,E1 -23097.078,E2 -23097.078} C_VEL
LIN {X 0,Y 184.437,Z 278.628,A -85,B 0,C 180,E1 -23099.042,E2 -23099.042} C_VEL
LIN {X 0,Y 183.874,Z 282.495,A -85,B 0,C 180,E1 -23100.206,E2 -23100.206} C_VEL
LIN {X 0,Y 180.675,Z 291.05,A -85,B 0,C 180,E1 -23102.803,E2 -23102.803} C_VEL
LIN {X 0,Y 177.518,Z 299.36,A -85,B 0,C 180,E1 -23106.044,E2 -23106.044} C_VEL
LIN {X 0,Y 175.03,Z 305.045,A -85,B 0,C 180,E1 -23108.815,E2 -23108.815} C_VEL
LIN {X 0,Y 172.664,Z 310.54,A -85,B 0,C 180,E1 -23112.226,E2 -23112.226} C_VEL
LIN {X 0,Y 170.927,Z 314.872,A -85,B 0,C 180,E1 -23115.718,E2 -23115.718} C_VEL
LIN {X 0,Y 170.089,Z 317.244,A -85,B 0,C 180,E1 -23118.077,E2 -23118.077} C_VEL
LIN {X 0,Y 169.482,Z 319.049,A -85,B 0,C 180,E1 -23120.452,E2 -23120.452} C_VEL
LIN {X 0,Y 168.934,Z 321.51,A -85,B 0,C 180,E1 -23125.227,E2 -23125.227} C_VEL
LIN {X 0,Y 168.89,Z 322.104,A -85,B 0,C 180,E1 -23127.615,E2 -23127.615} C_VEL
LIN {X 0,Y 168.965,Z 322.263,A -85,B 0,C 180,E1 -23130,E2 -23130} C_VEL
LIN {X 0,Y 168.877,Z 322.001,A -85,B 0,C 180,E1 -23132.801,E2 -23132.801} C_VEL
LIN {X 0,Y 168.934,Z 321.51,A -85,B 0,C 180,E1 -23134.773,E2 -23134.773} C_VEL
LIN {X 0,Y 169.483,Z 319.049,A -85,B 0,C 180,E1 -23139.548,E2 -23139.548} C_VEL
LIN {X 0,Y 170.481,Z 316.091,A -85,B 0,C 180,E1 -23143.105,E2 -23143.105} C_VEL
LIN {X 0,Y 171.961,Z 312.094,A -85,B 0,C 180,E1 -23146.624,E2 -23146.624} C_VEL
LIN {X 0,Y 174.223,Z 306.963,A -85,B 0,C 180,E1 -23150.052,E2 -23150.052} C_VEL
LIN {X 0,Y 176.483,Z 301.699,A -85,B 0,C 180,E1 -23152.847,E2 -23152.847} C_VEL
LIN {X 0,Y 178.442,Z 296.733,A -85,B 0,C 180,E1 -23155.058,E2 -23155.058} C_VEL
LIN {X 0,Y 181.267,Z 289.422,A -85,B 0,C 180,E1 -23157.726,E2 -23157.726} C_VEL
LIN {X 0,Y 183.876,Z 282.495,A -85,B 0,C 180,E1 -23159.793,E2 -23159.793} C_VEL
LIN {X 0,Y 184.661,Z 275.391,A -85,B 0,C 180,E1 -23161.874,E2 -23161.874} C_VEL
LIN {X 0,Y 184.797,Z 271.908,A -85,B 0,C 180,E1 -23162.828,E2 -23162.828} C_VEL
LIN {X 0,Y 184.324,Z 267.672,A -85,B 0,C 180,E1 -23164.094,E2 -23164.094} C_VEL
LIN {X 0,Y 182.852,Z 263.781,A -85,B 0,C 180,E1 -23165.422,E2 -23165.422} C_VEL
LIN {X 0,Y 178.884,Z 256.138,A -85,B 0,C 180,E1 -23168.089,E2 -23168.089} C_VEL
LIN {X 0,Y 177.31,Z 251.826,A -85,B 0,C 180,E1 -23169.338,E2 -23169.338} C_VEL
LIN {X 0,Y 176.961,Z 250.253,A -85,B 0,C 180,E1 -23169.723,E2 -23169.723} C_VEL
LIN {X 0,Y 174.582,Z 239.325,A -85,B 0,C 180,E1 -23172.351,E2 -23172.351} C_VEL
LIN {X 0,Y 171.618,Z 230.188,A -85,B 0,C 180,E1 -23174.637,E2 -23174.637} C_VEL
LIN {X 0,Y 169.66,Z 225.859,A -85,B 0,C 180,E1 -23175.805,E2 -23175.805} C_VEL
LIN {X 0,Y 167.661,Z 221.557,A -85,B 0,C 180,E1 -23177.037,E2 -23177.037} C_VEL
LIN {X 0,Y 165.837,Z 218.671,A -85,B 0,C 180,E1 -23177.991,E2 -23177.991} C_VEL
LIN {X 0,Y 165.242,Z 216.419,A -85,B 0,C 180,E1 -23178.487,E2 -23178.487} C_VEL
LIN {X 0,Y 164.993,Z 214.519,A -85,B 0,C 180,E1 -23183.39,E2 -23183.39} C_VEL
LIN {X 0,Y 164.782,Z 212.486,A -85,B 0,C 180,E1 -23189.215,E2 -23189.215} C_VEL
LIN {X 0,Y 164.58,Z 210.789,A -85,B 0,C 180,E1 -23194.72,E2 -23194.72} C_VEL
LIN {X 0,Y 164.485,Z 209.501,A -85,B 0,C 180,E1 -23200.049,E2 -23200.049} C_VEL
LIN {X 0,Y 164.504,Z 209.494,A -85,B 0,C 180,E1 -23205.146,E2 -23205.146} C_VEL
LIN {X 0,Y 164.767,Z 209.462,A -85,B 0,C 180,E1 -23210.175,E2 -23210.175} C_VEL
LIN {X 0,Y 164.829,Z 209.453,A -85,B 0,C 180,E1 -23212.65,E2 -23212.65} C_VEL
LIN {X 0,Y 165.045,Z 209.425,A -85,B 0,C 180,E1 -23217.558,E2 -23217.558} C_VEL
LIN {X 0,Y 165.293,Z 209.37,A -85,B 0,C 180,E1 -23219.999,E2 -23219.999} C_VEL
LIN {X 0,Y 164.759,Z 209.447,A -85,B 0,C 180,E1 -23224.893,E2 -23224.893} C_VEL
LIN {X 0,Y 164.828,Z 209.455,A -85,B 0,C 180,E1 -23227.348,E2 -23227.348} C_VEL
LIN {X 0,Y 164.7,Z 209.465,A -85,B 0,C 180,E1 -23231.06,E2 -23231.06} C_VEL
LIN {X 0,Y 164.481,Z 209.498,A -85,B 0,C 180,E1 -23237.402,E2 -23237.402} C_VEL
LIN {X 0,Y 164.471,Z 209.488,A -85,B 0,C 180,E1 -23239.988,E2 -23239.988} C_VEL
LIN {X 0,Y 164.385,Z 209.503,A -85,B 0,C 180,E1 -23246.129,E2 -23246.129} C_VEL
LIN {X 0,Y 164.373,Z 209.509,A -85,B 0,C 180,E1 -23251.227,E2 -23251.227} C_VEL
LIN {X 0,Y 164.31,Z 209.518,A -85,B 0,C 180,E1 -23256.784,E2 -23256.784} C_VEL
LIN {X 0,Y 164.34,Z 209.663,A -85,B 0,C 180,E1 -23261.21,E2 -23261.21} C_VEL
LIN {X 0,Y 165.185,Z 212.186,A -85,B 0,C 180,E1 -23261.766,E2 -23261.766} C_VEL
LIN {X 0,Y 167.463,Z 214.893,A -85,B 0,C 180,E1 -23262.906,E2 -23262.906} C_VEL
LIN {X 0,Y 169.416,Z 218.245,A -85,B 0,C 180,E1 -23264.038,E2 -23264.038} C_VEL
LIN {X 0,Y 170.69,Z 220.289,A -85,B 0,C 180,E1 -23264.732,E2 -23264.732} C_VEL
LIN {X 0,Y 174.868,Z 227.443,A -85,B 0,C 180,E1 -23267.091,E2 -23267.091} C_VEL
LIN {X 0,Y 179.023,Z 235.903,A -85,B 0,C 180,E1 -23269.686,E2 -23269.686} C_VEL
LIN {X 0,Y 182.368,Z 244.404,A -85,B 0,C 180,E1 -23272.183,E2 -23272.183} C_VEL
LIN {X 0,Y 185.376,Z 253.823,A -85,B 0,C 180,E1 -23274.995,E2 -23274.995} C_VEL
LIN {X 0,Y 187.253,Z 262.296,A -85,B 0,C 180,E1 -23277.574,E2 -23277.574} C_VEL
LIN {X 0,Y 189.428,Z 270.442,A -85,B 0,C 180,E1 -23280.396,E2 -23280.396} C_VEL
LIN {X 0,Y 191.73,Z 276.378,A -85,B 0,C 180,E1 -23282.742,E2 -23282.742} C_VEL
LIN {X 0,Y 196.196,Z 284.065,A -85,B 0,C 180,E1 -23286.313,E2 -23286.313} C_VEL
LIN {X 0,Y 201.375,Z 290.116,A -85,B 0,C 180,E1 -23289.574,E2 -23289.574} C_VEL
LIN {X 0,Y 206.541,Z 294.624,A -85,B 0,C 180,E1 -23292.315,E2 -23292.315} C_VEL
LIN {X 0,Y 213.943,Z 299.456,A -85,B 0,C 180,E1 -23295.708,E2 -23295.708} C_VEL
LIN {X 0,Y 222.334,Z 303.482,A -85,B 0,C 180,E1 -23299.067,E2 -23299.067} C_VEL
LIN {X 0,Y 227.874,Z 305.588,A -85,B 0,C 180,E1 -23301.129,E2 -23301.129} C_VEL
LIN {X 0,Y 233.564,Z 307.31,A -85,B 0,C 180,E1 -23303.196,E2 -23303.196} C_VEL
LIN {X 0,Y 239.657,Z 308.822,A -85,B 0,C 180,E1 -23305.591,E2 -23305.591} C_VEL
LIN {X 0,Y 241.958,Z 309.332,A -85,B 0,C 180,E1 -23306.67,E2 -23306.67} C_VEL
LIN {X 0,Y 246.014,Z 309.906,A -85,B 0,C 180,E1 -23308.984,E2 -23308.984} C_VEL
LIN {X 0,Y 247.163,Z 309.931,A -85,B 0,C 180,E1 -23310,E2 -23310} C_VEL
LIN {X 0,Y 246.014,Z 309.906,A -85,B 0,C 180,E1 -23311.016,E2 -23311.016} C_VEL
LIN {X 0,Y 241.956,Z 309.331,A -85,B 0,C 180,E1 -23313.33,E2 -23313.33} C_VEL
LIN {X 0,Y 237.994,Z 308.433,A -85,B 0,C 180,E1 -23315.082,E2 -23315.082} C_VEL
LIN {X 0,Y 233.248,Z 307.222,A -85,B 0,C 180,E1 -23316.922,E2 -23316.922} C_VEL
LIN {X 0,Y 225.1,Z 304.587,A -85,B 0,C 180,E1 -23319.887,E2 -23319.887} C_VEL
LIN {X 0,Y 216.539,Z 300.865,A -85,B 0,C 180,E1 -23323.18,E2 -23323.18} C_VEL
LIN {X 0,Y 208.907,Z 296.298,A -85,B 0,C 180,E1 -23326.541,E2 -23326.541} C_VEL
LIN {X 0,Y 202.01,Z 290.727,A -85,B 0,C 180,E1 -23330.062,E2 -23330.062} C_VEL
LIN {X 0,Y 197.032,Z 285.199,A -85,B 0,C 180,E1 -23333.101,E2 -23333.101} C_VEL
LIN {X 0,Y 193.322,Z 279.486,A -85,B 0,C 180,E1 -23335.864,E2 -23335.864} C_VEL
LIN {X 0,Y 190.261,Z 272.792,A -85,B 0,C 180,E1 -23338.698,E2 -23338.698} C_VEL
LIN {X 0,Y 188.143,Z 266.16,A -85,B 0,C 180,E1 -23341.157,E2 -23341.157} C_VEL
LIN {X 0,Y 186.25,Z 257.568,A -85,B 0,C 180,E1 -23343.888,E2 -23343.888} C_VEL
LIN {X 0,Y 184.398,Z 250.452,A -85,B 0,C 180,E1 -23346.033,E2 -23346.033} C_VEL
LIN {X 0,Y 181.684,Z 242.293,A -85,B 0,C 180,E1 -23348.437,E2 -23348.437} C_VEL
LIN {X 0,Y 177.646,Z 232.79,A -85,B 0,C 180,E1 -23351.267,E2 -23351.267} C_VEL
LIN {X 0,Y 171.901,Z 222.154,A -85,B 0,C 180,E1 -23354.634,E2 -23354.634} C_VEL
LIN {X 0,Y 169.559,Z 218.394,A -85,B 0,C 180,E1 -23355.893,E2 -23355.893} C_VEL
LIN {X 0,Y 167.547,Z 215.162,A -85,B 0,C 180,E1 -23357.028,E2 -23357.028} C_VEL
LIN {X 0,Y 167.044,Z 214.264,A -85,B 0,C 180,E1 -23357.326,E2 -23357.326} C_VEL
LIN {X 0,Y 165.092,Z 211.959,A -85,B 0,C 180,E1 -23358.307,E2 -23358.307} C_VEL
LIN {X 0,Y 164.309,Z 209.517,A -85,B 0,C 180,E1 -23358.882,E2 -23358.882} C_VEL
LIN {X 0,Y 164.34,Z 209.513,A -85,B 0,C 180,E1 -23364.343,E2 -23364.343} C_VEL
LIN {X 0,Y 164.388,Z 209.507,A -85,B 0,C 180,E1 -23369.136,E2 -23369.136} C_VEL
LIN {X 0,Y 164.407,Z 209.497,A -85,B 0,C 180,E1 -23374.694,E2 -23374.694} C_VEL
LIN {X 0,Y 164.482,Z 209.486,A -85,B 0,C 180,E1 -23380.052,E2 -23380.052} C_VEL
LIN {X 0,Y 164.503,Z 209.485,A -85,B 0,C 180,E1 -23385.149,E2 -23385.149} C_VEL
LIN {X 0,Y 164.765,Z 209.452,A -85,B 0,C 180,E1 -23390.178,E2 -23390.178} C_VEL
LIN {X 0,Y 164.828,Z 209.455,A -85,B 0,C 180,E1 -23392.652,E2 -23392.652} C_VEL
LIN {X 0,Y 165.044,Z 209.389,A -85,B 0,C 180,E1 -23397.561,E2 -23397.561} C_VEL
LIN {X 0,Y 165.293,Z 209.37,A -85,B 0,C 180,E1 -23400.001,E2 -23400.001} C_VEL
LIN {X 0,Y 164.761,Z 209.462,A -85,B 0,C 180,E1 -23404.895,E2 -23404.895} C_VEL
LIN {X 0,Y 164.829,Z 209.454,A -85,B 0,C 180,E1 -23407.35,E2 -23407.35} C_VEL
LIN {X 0,Y 164.702,Z 209.47,A -85,B 0,C 180,E1 -23411.062,E2 -23411.062} C_VEL
LIN {X 0,Y 164.483,Z 209.497,A -85,B 0,C 180,E1 -23417.405,E2 -23417.405} C_VEL
LIN {X 0,Y 164.474,Z 209.499,A -85,B 0,C 180,E1 -23419.99,E2 -23419.99} C_VEL
LIN {X 0,Y 164.633,Z 211.097,A -85,B 0,C 180,E1 -23426.304,E2 -23426.304} C_VEL
LIN {X 0,Y 164.805,Z 212.726,A -85,B 0,C 180,E1 -23431.474,E2 -23431.474} C_VEL
LIN {X 0,Y 164.995,Z 214.518,A -85,B 0,C 180,E1 -23436.609,E2 -23436.609} C_VEL
LIN {X 0,Y 165.236,Z 216.515,A -85,B 0,C 180,E1 -23441.564,E2 -23441.564} C_VEL
LIN {X 0,Y 166.399,Z 219.849,A -85,B 0,C 180,E1 -23442.321,E2 -23442.321} C_VEL
LIN {X 0,Y 168.189,Z 222.42,A -85,B 0,C 180,E1 -23443.26,E2 -23443.26} C_VEL
LIN {X 0,Y 169.996,Z 226.356,A -85,B 0,C 180,E1 -23444.369,E2 -23444.369} C_VEL
LIN {X 0,Y 172.923,Z 233.751,A -85,B 0,C 180,E1 -23446.298,E2 -23446.298} C_VEL
LIN {X 0,Y 175.517,Z 243.079,A -85,B 0,C 180,E1 -23448.555,E2 -23448.555} C_VEL
LIN {X 0,Y 177.388,Z 253.054,A -85,B 0,C 180,E1 -23450.983,E2 -23450.983} C_VEL
LIN {X 0,Y 178.291,Z 262.173,A -85,B 0,C 180,E1 -23453.274,E2 -23453.274} C_VEL
LIN {X 0,Y 178.47,Z 271.474,A -85,B 0,C 180,E1 -23455.79,E2 -23455.79} C_VEL
LIN {X 0,Y 178.033,Z 278.404,A -85,B 0,C 180,E1 -23457.797,E2 -23457.797} C_VEL
LIN {X 0,Y 177.555,Z 282.277,A -85,B 0,C 180,E1 -23459.032,E2 -23459.032} C_VEL
LIN {X 0,Y 175.698,Z 287.584,A -85,B 0,C 180,E1 -23460.66,E2 -23460.66} C_VEL
LIN {X 0,Y 173.149,Z 293.787,A -85,B 0,C 180,E1 -23462.831,E2 -23462.831} C_VEL
LIN {X 0,Y 170.465,Z 300.331,A -85,B 0,C 180,E1 -23465.652,E2 -23465.652} C_VEL
LIN {X 0,Y 168.388,Z 304.832,A -85,B 0,C 180,E1 -23467.937,E2 -23467.937} C_VEL
LIN {X 0,Y 165.9,Z 310.328,A -85,B 0,C 180,E1 -23471.475,E2 -23471.475} C_VEL
LIN {X 0,Y 164.003,Z 314.659,A -85,B 0,C 180,E1 -23475.101,E2 -23475.101} C_VEL
LIN {X 0,Y 163.133,Z 317.032,A -85,B 0,C 180,E1 -23477.561,E2 -23477.561} C_VEL
LIN {X 0,Y 162.456,Z 318.837,A -85,B 0,C 180,E1 -23480.035,E2 -23480.035} C_VEL
LIN {X 0,Y 161.854,Z 321.298,A -85,B 0,C 180,E1 -23485.018,E2 -23485.018} C_VEL
LIN {X 0,Y 161.8,Z 321.893,A -85,B 0,C 180,E1 -23487.511,E2 -23487.511} C_VEL
LIN {X 0,Y 161.884,Z 322.053,A -85,B 0,C 180,E1 -23490,E2 -23490} C_VEL
LIN {X 0,Y 161.8,Z 321.893,A -85,B 0,C 180,E1 -23492.489,E2 -23492.489} C_VEL
LIN {X 0,Y 161.854,Z 321.298,A -85,B 0,C 180,E1 -23494.982,E2 -23494.982} C_VEL
LIN {X 0,Y 162.457,Z 318.837,A -85,B 0,C 180,E1 -23499.965,E2 -23499.965} C_VEL
LIN {X 0,Y 163.531,Z 315.879,A -85,B 0,C 180,E1 -23503.672,E2 -23503.672} C_VEL
LIN {X 0,Y 165.147,Z 311.882,A -85,B 0,C 180,E1 -23507.331,E2 -23507.331} C_VEL
LIN {X 0,Y 167.545,Z 306.751,A -85,B 0,C 180,E1 -23510.888,E2 -23510.888} C_VEL
LIN {X 0,Y 169.95,Z 301.488,A -85,B 0,C 180,E1 -23513.778,E2 -23513.778} C_VEL
LIN {X 0,Y 171.789,Z 297.081,A -85,B 0,C 180,E1 -23515.835,E2 -23515.835} C_VEL
LIN {X 0,Y 174.342,Z 290.837,A -85,B 0,C 180,E1 -23518.272,E2 -23518.272} C_VEL
LIN {X 0,Y 177.048,Z 284.204,A -85,B 0,C 180,E1 -23520.405,E2 -23520.405} C_VEL
LIN {X 0,Y 177.833,Z 280.342,A -85,B 0,C 180,E1 -23521.576,E2 -23521.576} C_VEL
LIN {X 0,Y 178.394,Z 272.582,A -85,B 0,C 180,E1 -23523.897,E2 -23523.897} C_VEL
LIN {X 0,Y 178.366,Z 264.039,A -85,B 0,C 180,E1 -23526.23,E2 -23526.23} C_VEL
LIN {X 0,Y 177.764,Z 256.233,A -85,B 0,C 180,E1 -23528.224,E2 -23528.224} C_VEL
LIN {X 0,Y 176.961,Z 250.253,A -85,B 0,C 180,E1 -23529.723,E2 -23529.723} C_VEL
LIN {X 0,Y 175.548,Z 245.855,A -85,B 0,C 180,E1 -23530.919,E2 -23530.919} C_VEL
LIN {X 0,Y 173.385,Z 242.069,A -85,B 0,C 180,E1 -23532.248,E2 -23532.248} C_VEL
LIN {X 0,Y 166.401,Z 232.801,A -85,B 0,C 180,E1 -23536.013,E2 -23536.013} C_VEL
LIN {X 0,Y 164.964,Z 230.137,A -85,B 0,C 180,E1 -23536.932,E2 -23536.932} C_VEL
LIN {X 0,Y 163.158,Z 226.295,A -85,B 0,C 180,E1 -23538.112,E2 -23538.112} C_VEL
LIN {X 0,Y 161.387,Z 222.795,A -85,B 0,C 180,E1 -23539.279,E2 -23539.279} C_VEL
LIN {X 0,Y 160.809,Z 221.525,A -85,B 0,C 180,E1 -23539.69,E2 -23539.69} C_VEL
LIN {X 0,Y 158.781,Z 218.635,A -85,B 0,C 180,E1 -23540.874,E2 -23540.874} C_VEL
LIN {X 0,Y 158.01,Z 216.118,A -85,B 0,C 180,E1 -23541.485,E2 -23541.485} C_VEL
LIN {X 0,Y 157.87,Z 215,A -85,B 0,C 180,E1 -23544.637,E2 -23544.637} C_VEL
LIN {X 0,Y 157.748,Z 213.955,A -85,B 0,C 180,E1 -23547.831,E2 -23547.831} C_VEL
LIN {X 0,Y 157.597,Z 212.244,A -85,B 0,C 180,E1 -23553.515,E2 -23553.515} C_VEL
LIN {X 0,Y 157.444,Z 210.668,A -85,B 0,C 180,E1 -23559.617,E2 -23559.617} C_VEL
LIN {X 0,Y 157.441,Z 210.374,A -85,B 0,C 180,E1 -23564.463,E2 -23564.463} C_VEL
LIN {X 0,Y 157.688,Z 210.344,A -85,B 0,C 180,E1 -23569.729,E2 -23569.729} C_VEL
LIN {X 0,Y 157.766,Z 210.333,A -85,B 0,C 180,E1 -23572.319,E2 -23572.319} C_VEL
LIN {X 0,Y 158.255,Z 210.245,A -85,B 0,C 180,E1 -23579.999,E2 -23579.999} C_VEL
LIN {X 0,Y 157.765,Z 210.333,A -85,B 0,C 180,E1 -23587.679,E2 -23587.679} C_VEL
LIN {X 0,Y 157.635,Z 210.345,A -85,B 0,C 180,E1 -23591.236,E2 -23591.236} C_VEL
LIN {X 0,Y 157.44,Z 210.366,A -85,B 0,C 180,E1 -23595.534,E2 -23595.534} C_VEL
LIN {X 0,Y 157.367,Z 210.375,A -85,B 0,C 180,E1 -23600.932,E2 -23600.932} C_VEL
LIN {X 0,Y 157.308,Z 210.388,A -85,B 0,C 180,E1 -23606.681,E2 -23606.681} C_VEL
LIN {X 0,Y 157.275,Z 210.395,A -85,B 0,C 180,E1 -23612.426,E2 -23612.426} C_VEL
LIN {X 0,Y 157.253,Z 210.397,A -85,B 0,C 180,E1 -23617.475,E2 -23617.475} C_VEL
LIN {X 0,Y 157.213,Z 210.413,A -85,B 0,C 180,E1 -23618.19,E2 -23618.19} C_VEL
LIN {X 0,Y 158.026,Z 212.869,A -85,B 0,C 180,E1 -23618.804,E2 -23618.804} C_VEL
LIN {X 0,Y 159.995,Z 215.166,A -85,B 0,C 180,E1 -23619.937,E2 -23619.937} C_VEL
LIN {X 0,Y 160.685,Z 216.12,A -85,B 0,C 180,E1 -23620.368,E2 -23620.368} C_VEL
LIN {X 0,Y 162.532,Z 219.259,A -85,B 0,C 180,E1 -23621.564,E2 -23621.564} C_VEL
LIN {X 0,Y 163.682,Z 220.883,A -85,B 0,C 180,E1 -23622.237,E2 -23622.237} C_VEL
LIN {X 0,Y 167.614,Z 227.472,A -85,B 0,C 180,E1 -23624.695,E2 -23624.695} C_VEL
LIN {X 0,Y 171.729,Z 235.475,A -85,B 0,C 180,E1 -23627.445,E2 -23627.445} C_VEL
LIN {X 0,Y 175.47,Z 244.399,A -85,B 0,C 180,E1 -23630.352,E2 -23630.352} C_VEL
LIN {X 0,Y 178.438,Z 253.711,A -85,B 0,C 180,E1 -23633.323,E2 -23633.323} C_VEL
LIN {X 0,Y 180.512,Z 262.632,A -85,B 0,C 180,E1 -23636.235,E2 -23636.235} C_VEL
LIN {X 0,Y 182.265,Z 270.866,A -85,B 0,C 180,E1 -23639.171,E2 -23639.171} C_VEL
LIN {X 0,Y 184.705,Z 278.051,A -85,B 0,C 180,E1 -23642.172,E2 -23642.172} C_VEL
LIN {X 0,Y 187.858,Z 283.963,A -85,B 0,C 180,E1 -23645.031,E2 -23645.031} C_VEL
LIN {X 0,Y 191.867,Z 289.536,A -85,B 0,C 180,E1 -23648.076,E2 -23648.076} C_VEL
LIN {X 0,Y 197.151,Z 294.642,A -85,B 0,C 180,E1 -23651.287,E2 -23651.287} C_VEL
LIN {X 0,Y 203.951,Z 299.416,A -85,B 0,C 180,E1 -23654.761,E2 -23654.761} C_VEL
LIN {X 0,Y 212.807,Z 303.765,A -85,B 0,C 180,E1 -23658.571,E2 -23658.571} C_VEL
LIN {X 0,Y 220.306,Z 306.46,A -85,B 0,C 180,E1 -23661.46,E2 -23661.46} C_VEL
LIN {X 0,Y 226.284,Z 308.096,A -85,B 0,C 180,E1 -23663.639,E2 -23663.639} C_VEL
LIN {X 0,Y 233.759,Z 309.578,A -85,B 0,C 180,E1 -23666.553,E2 -23666.553} C_VEL
LIN {X 0,Y 237.136,Z 310.048,A -85,B 0,C 180,E1 -23668.302,E2 -23668.302} C_VEL
LIN {X 0,Y 238.964,Z 310.155,A -85,B 0,C 180,E1 -23669.335,E2 -23669.335} C_VEL
LIN {X 0,Y 239.832,Z 310.145,A -85,B 0,C 180,E1 -23670,E2 -23670} C_VEL
LIN {X 0,Y 238.964,Z 310.155,A -85,B 0,C 180,E1 -23670.665,E2 -23670.665} C_VEL
LIN {X 0,Y 237.134,Z 310.048,A -85,B 0,C 180,E1 -23671.698,E2 -23671.698} C_VEL
LIN {X 0,Y 233.764,Z 309.577,A -85,B 0,C 180,E1 -23673.447,E2 -23673.447} C_VEL
LIN {X 0,Y 226.285,Z 308.094,A -85,B 0,C 180,E1 -23676.363,E2 -23676.363} C_VEL
LIN {X 0,Y 218.37,Z 305.875,A -85,B 0,C 180,E1 -23679.26,E2 -23679.26} C_VEL
LIN {X 0,Y 209.11,Z 302.196,A -85,B 0,C 180,E1 -23682.93,E2 -23682.93} C_VEL
LIN {X 0,Y 200.561,Z 297.2,A -85,B 0,C 180,E1 -23686.888,E2 -23686.888} C_VEL
LIN {X 0,Y 194.651,Z 292.378,A -85,B 0,C 180,E1 -23690.161,E2 -23690.161} C_VEL
LIN {X 0,Y 190.601,Z 288.018,A -85,B 0,C 180,E1 -23692.809,E2 -23692.809} C_VEL
LIN {X 0,Y 185.888,Z 280.557,A -85,B 0,C 180,E1 -23696.664,E2 -23696.664} C_VEL
LIN {X 0,Y 183.476,Z 274.783,A -85,B 0,C 180,E1 -23699.273,E2 -23699.273} C_VEL
LIN {X 0,Y 181.315,Z 266.922,A -85,B 0,C 180,E1 -23702.314,E2 -23702.314} C_VEL
LIN {X 0,Y 179.588,Z 258.207,A -85,B 0,C 180,E1 -23705.225,E2 -23705.225} C_VEL
LIN {X 0,Y 177.211,Z 249.643,A -85,B 0,C 180,E1 -23707.983,E2 -23707.983} C_VEL
LIN {X 0,Y 174.052,Z 240.876,A -85,B 0,C 180,E1 -23710.793,E2 -23710.793} C_VEL
LIN {X 0,Y 170.093,Z 232.152,A -85,B 0,C 180,E1 -23713.693,E2 -23713.693} C_VEL
LIN {X 0,Y 166.045,Z 224.592,A -85,B 0,C 180,E1 -23716.359,E2 -23716.359} C_VEL
LIN {X 0,Y 163.367,Z 220.221,A -85,B 0,C 180,E1 -23717.974,E2 -23717.974} C_VEL
LIN {X 0,Y 161.028,Z 216.93,A -85,B 0,C 180,E1 -23719.374,E2 -23719.374} C_VEL
LIN {X 0,Y 160.247,Z 215.351,A -85,B 0,C 180,E1 -23719.928,E2 -23719.928} C_VEL
LIN {X 0,Y 158.145,Z 213.075,A -85,B 0,C 180,E1 -23721.131,E2 -23721.131} C_VEL
LIN {X 0,Y 157.222,Z 210.399,A -85,B 0,C 180,E1 -23721.891,E2 -23721.891} C_VEL
LIN {X 0,Y 157.287,Z 210.391,A -85,B 0,C 180,E1 -23724.49,E2 -23724.49} C_VEL
LIN {X 0,Y 157.291,Z 210.392,A -85,B 0,C 180,E1 -23728.096,E2 -23728.096} C_VEL
LIN {X 0,Y 157.315,Z 210.386,A -85,B 0,C 180,E1 -23733.466,E2 -23733.466} C_VEL
LIN {X 0,Y 157.391,Z 210.37,A -85,B 0,C 180,E1 -23739.669,E2 -23739.669} C_VEL
LIN {X 0,Y 157.44,Z 210.366,A -85,B 0,C 180,E1 -23744.466,E2 -23744.466} C_VEL
LIN {X 0,Y 157.687,Z 210.334,A -85,B 0,C 180,E1 -23749.732,E2 -23749.732} C_VEL
LIN {X 0,Y 157.765,Z 210.333,A -85,B 0,C 180,E1 -23752.321,E2 -23752.321} C_VEL
LIN {X 0,Y 158.255,Z 210.245,A -85,B 0,C 180,E1 -23760.001,E2 -23760.001} C_VEL
LIN {X 0,Y 157.766,Z 210.335,A -85,B 0,C 180,E1 -23767.681,E2 -23767.681} C_VEL
LIN {X 0,Y 157.636,Z 210.35,A -85,B 0,C 180,E1 -23771.238,E2 -23771.238} C_VEL
LIN {X 0,Y 157.441,Z 210.376,A -85,B 0,C 180,E1 -23775.537,E2 -23775.537} C_VEL
LIN {X 0,Y 157.444,Z 210.664,A -85,B 0,C 180,E1 -23780.383,E2 -23780.383} C_VEL
LIN {X 0,Y 157.622,Z 212.237,A -85,B 0,C 180,E1 -23786.481,E2 -23786.481} C_VEL
LIN {X 0,Y 157.763,Z 214,A -85,B 0,C 180,E1 -23792.316,E2 -23792.316} C_VEL
LIN {X 0,Y 157.957,Z 215.523,A -85,B 0,C 180,E1 -23796.787,E2 -23796.787} C_VEL
LIN {X 0,Y 158.052,Z 216.291,A -85,B 0,C 180,E1 -23798.572,E2 -23798.572} C_VEL
LIN {X 0,Y 159.086,Z 219.243,A -85,B 0,C 180,E1 -23799.317,E2 -23799.317} C_VEL
LIN {X 0,Y 161.27,Z 222.453,A -85,B 0,C 180,E1 -23800.626,E2 -23800.626} C_VEL
LIN {X 0,Y 162.92,Z 225.99,A -85,B 0,C 180,E1 -23801.756,E2 -23801.756} C_VEL
LIN {X 0,Y 164.025,Z 228.023,A -85,B 0,C 180,E1 -23802.444,E2 -23802.444} C_VEL
LIN {X 0,Y 166.751,Z 234.508,A -85,B 0,C 180,E1 -23804.404,E2 -23804.404} C_VEL
LIN {X 0,Y 169.161,Z 242.454,A -85,B 0,C 180,E1 -23806.551,E2 -23806.551} C_VEL
LIN {X 0,Y 170.984,Z 251.888,A -85,B 0,C 180,E1 -23809.005,E2 -23809.005} C_VEL
LIN {X 0,Y 171.983,Z 261.936,A -85,B 0,C 180,E1 -23811.69,E2 -23811.69} C_VEL
LIN {X 0,Y 172.165,Z 270.352,A -85,B 0,C 180,E1 -23814.071,E2 -23814.071} C_VEL
LIN {X 0,Y 171.731,Z 278.181,A -85,B 0,C 180,E1 -23816.463,E2 -23816.463} C_VEL
LIN {X 0,Y 170.858,Z 283.989,A -85,B 0,C 180,E1 -23818.369,E2 -23818.369} C_VEL
LIN {X 0,Y 166.84,Z 293.575,A -85,B 0,C 180,E1 -23821.713,E2 -23821.713} C_VEL
LIN {X 0,Y 163.969,Z 300.118,A -85,B 0,C 180,E1 -23824.621,E2 -23824.621} C_VEL
LIN {X 0,Y 161.803,Z 304.62,A -85,B 0,C 180,E1 -23826.989,E2 -23826.989} C_VEL
LIN {X 0,Y 159.171,Z 310.116,A -85,B 0,C 180,E1 -23830.661,E2 -23830.661} C_VEL
LIN {X 0,Y 157.103,Z 314.446,A -85,B 0,C 180,E1 -23834.431,E2 -23834.431} C_VEL
LIN {X 0,Y 156.176,Z 316.82,A -85,B 0,C 180,E1 -23836.997,E2 -23836.997} C_VEL
LIN {X 0,Y 155.453,Z 318.625,A -85,B 0,C 180,E1 -23839.582,E2 -23839.582} C_VEL
LIN {X 0,Y 154.76,Z 321.086,A -85,B 0,C 180,E1 -23844.789,E2 -23844.789} C_VEL
LIN {X 0,Y 154.715,Z 321.803,A -85,B 0,C 180,E1 -23847.983,E2 -23847.983} C_VEL
LIN {X 0,Y 154.715,Z 321.803,A -85,B 0,C 180,E1 -23852.017,E2 -23852.017} C_VEL
LIN {X 0,Y 154.76,Z 321.086,A -85,B 0,C 180,E1 -23855.211,E2 -23855.211} C_VEL
LIN {X 0,Y 155.453,Z 318.625,A -85,B 0,C 180,E1 -23860.418,E2 -23860.418} C_VEL
LIN {X 0,Y 156.604,Z 315.666,A -85,B 0,C 180,E1 -23864.29,E2 -23864.29} C_VEL
LIN {X 0,Y 158.367,Z 311.67,A -85,B 0,C 180,E1 -23868.098,E2 -23868.098} C_VEL
LIN {X 0,Y 160.89,Z 306.538,A -85,B 0,C 180,E1 -23871.795,E2 -23871.795} C_VEL
LIN {X 0,Y 163.447,Z 301.275,A -85,B 0,C 180,E1 -23874.786,E2 -23874.786} C_VEL
LIN {X 0,Y 166.222,Z 294.952,A -85,B 0,C 180,E1 -23877.716,E2 -23877.716} C_VEL
LIN {X 0,Y 168.773,Z 288.997,A -85,B 0,C 180,E1 -23879.98,E2 -23879.98} C_VEL
LIN {X 0,Y 170.861,Z 283.989,A -85,B 0,C 180,E1 -23881.63,E2 -23881.63} C_VEL
LIN {X 0,Y 171.897,Z 276.086,A -85,B 0,C 180,E1 -23884.205,E2 -23884.205} C_VEL
LIN {X 0,Y 172.181,Z 266.548,A -85,B 0,C 180,E1 -23887.016,E2 -23887.016} C_VEL
LIN {X 0,Y 171.704,Z 257.828,A -85,B 0,C 180,E1 -23889.413,E2 -23889.413} C_VEL
LIN {X 0,Y 170.294,Z 247.906,A -85,B 0,C 180,E1 -23892.023,E2 -23892.023} C_VEL
LIN {X 0,Y 168.257,Z 239.02,A -85,B 0,C 180,E1 -23894.354,E2 -23894.354} C_VEL
LIN {X 0,Y 165.78,Z 231.899,A -85,B 0,C 180,E1 -23896.373,E2 -23896.373} C_VEL
LIN {X 0,Y 164.964,Z 230.137,A -85,B 0,C 180,E1 -23896.932,E2 -23896.932} C_VEL
LIN {X 0,Y 163.384,Z 227.735,A -85,B 0,C 180,E1 -23897.878,E2 -23897.878} C_VEL
LIN {X 0,Y 159.912,Z 224.997,A -85,B 0,C 180,E1 -23899.63,E2 -23899.63} C_VEL
LIN {X 0,Y 153.981,Z 221.57,A -85,B 0,C 180,E1 -23902.728,E2 -23902.728} C_VEL
LIN {X 0,Y 151.853,Z 218.92,A -85,B 0,C 180,E1 -23904.142,E2 -23904.142} C_VEL
LIN {X 0,Y 150.791,Z 215.77,A -85,B 0,C 180,E1 -23905.081,E2 -23905.081} C_VEL
LIN {X 0,Y 150.652,Z 214.538,A -85,B 0,C 180,E1 -23909.124,E2 -23909.124} C_VEL
LIN {X 0,Y 150.575,Z 213.584,A -85,B 0,C 180,E1 -23912.474,E2 -23912.474} C_VEL
LIN {X 0,Y 150.397,Z 212.17,A -85,B 0,C 180,E1 -23918.046,E2 -23918.046} C_VEL
LIN {X 0,Y 150.379,Z 211.519,A -85,B 0,C 180,E1 -23920.903,E2 -23920.903} C_VEL
LIN {X 0,Y 150.429,Z 211.248,A -85,B 0,C 180,E1 -23926.49,E2 -23926.49} C_VEL
LIN {X 0,Y 150.61,Z 211.225,A -85,B 0,C 180,E1 -23929.241,E2 -23929.241} C_VEL
LIN {X 0,Y 150.703,Z 211.214,A -85,B 0,C 180,E1 -23931.956,E2 -23931.956} C_VEL
LIN {X 0,Y 151.215,Z 211.119,A -85,B 0,C 180,E1 -23939.999,E2 -23939.999} C_VEL
LIN {X 0,Y 150.702,Z 211.211,A -85,B 0,C 180,E1 -23948.041,E2 -23948.041} C_VEL
LIN {X 0,Y 150.575,Z 211.226,A -85,B 0,C 180,E1 -23951.436,E2 -23951.436} C_VEL
LIN {X 0,Y 150.351,Z 211.252,A -85,B 0,C 180,E1 -23956.286,E2 -23956.286} C_VEL
LIN {X 0,Y 150.348,Z 211.248,A -85,B 0,C 180,E1 -23960.791,E2 -23960.791} C_VEL
LIN {X 0,Y 150.239,Z 211.272,A -85,B 0,C 180,E1 -23967.279,E2 -23967.279} C_VEL
LIN {X 0,Y 150.215,Z 211.274,A -85,B 0,C 180,E1 -23972.633,E2 -23972.633} C_VEL
LIN {X 0,Y 150.206,Z 211.328,A -85,B 0,C 180,E1 -23974.714,E2 -23974.714} C_VEL
LIN {X 0,Y 151.064,Z 213.786,A -85,B 0,C 180,E1 -23975.455,E2 -23975.455} C_VEL
LIN {X 0,Y 152.866,Z 215.963,A -85,B 0,C 180,E1 -23976.702,E2 -23976.702} C_VEL
LIN {X 0,Y 153.76,Z 216.952,A -85,B 0,C 180,E1 -23977.308,E2 -23977.308} C_VEL
LIN {X 0,Y 155.396,Z 219.919,A -85,B 0,C 180,E1 -23978.552,E2 -23978.552} C_VEL
LIN {X 0,Y 156.931,Z 221.898,A -85,B 0,C 180,E1 -23979.55,E2 -23979.55} C_VEL
LIN {X 0,Y 161.881,Z 230.205,A -85,B 0,C 180,E1 -23983.053,E2 -23983.053} C_VEL
LIN {X 0,Y 165.868,Z 238.159,A -85,B 0,C 180,E1 -23986.078,E2 -23986.078} C_VEL
LIN {X 0,Y 168.771,Z 245.105,A -85,B 0,C 180,E1 -23988.55,E2 -23988.55} C_VEL
LIN {X 0,Y 171.899,Z 254.756,A -85,B 0,C 180,E1 -23991.906,E2 -23991.906} C_VEL
LIN {X 0,Y 173.69,Z 262.332,A -85,B 0,C 180,E1 -23994.542,E2 -23994.542} C_VEL
LIN {X 0,Y 175.28,Z 271.31,A -85,B 0,C 180,E1 -23997.872,E2 -23997.872} C_VEL
LIN {X 0,Y 177.153,Z 278.068,A -85,B 0,C 180,E1 -24000.78,E2 -24000.78} C_VEL
LIN {X 0,Y 179.944,Z 284.392,A -85,B 0,C 180,E1 -24003.933,E2 -24003.933} C_VEL
LIN {X 0,Y 184.113,Z 290.656,A -85,B 0,C 180,E1 -24007.56,E2 -24007.56} C_VEL
LIN {X 0,Y 189.557,Z 296.002,A -85,B 0,C 180,E1 -24011.181,E2 -24011.181} C_VEL
LIN {X 0,Y 196.493,Z 300.755,A -85,B 0,C 180,E1 -24014.948,E2 -24014.948} C_VEL
LIN {X 0,Y 203.253,Z 304.05,A -85,B 0,C 180,E1 -24018.026,E2 -24018.026} C_VEL
LIN {X 0,Y 212.961,Z 307.352,A -85,B 0,C 180,E1 -24021.899,E2 -24021.899} C_VEL
LIN {X 0,Y 220.03,Z 308.962,A -85,B 0,C 180,E1 -24024.501,E2 -24024.501} C_VEL
LIN {X 0,Y 225.312,Z 309.861,A -85,B 0,C 180,E1 -24026.499,E2 -24026.499} C_VEL
LIN {X 0,Y 229.149,Z 310.285,A -85,B 0,C 180,E1 -24028.242,E2 -24028.242} C_VEL
LIN {X 0,Y 232.396,Z 310.362,A -85,B 0,C 180,E1 -24030,E2 -24030} C_VEL
LIN {X 0,Y 229.15,Z 310.285,A -85,B 0,C 180,E1 -24031.757,E2 -24031.757} C_VEL
LIN {X 0,Y 225.109,Z 309.836,A -85,B 0,C 180,E1 -24033.58,E2 -24033.58} C_VEL
LIN {X 0,Y 219.011,Z 308.777,A -85,B 0,C 180,E1 -24035.867,E2 -24035.867} C_VEL
LIN {X 0,Y 212.96,Z 307.354,A -85,B 0,C 180,E1 -24038.099,E2 -24038.099} C_VEL
LIN {X 0,Y 203.203,Z 304.052,A -85,B 0,C 180,E1 -24041.977,E2 -24041.977} C_VEL
LIN {X 0,Y 194.3,Z 299.474,A -85,B 0,C 180,E1 -24046.181,E2 -24046.181} C_VEL
LIN {X 0,Y 186.267,Z 293.026,A -85,B 0,C 180,E1 -24050.912,E2 -24050.912} C_VEL
LIN {X 0,Y 181.492,Z 286.996,A -85,B 0,C 180,E1 -24054.619,E2 -24054.619} C_VEL
LIN {X 0,Y 178.515,Z 281.506,A -85,B 0,C 180,E1 -24057.576,E2 -24057.576} C_VEL
LIN {X 0,Y 176.229,Z 275.021,A -85,B 0,C 180,E1 -24060.605,E2 -24060.605} C_VEL
LIN {X 0,Y 174.542,Z 267.253,A -85,B 0,C 180,E1 -24063.703,E2 -24063.703} C_VEL
LIN {X 0,Y 172.826,Z 258.395,A -85,B 0,C 180,E1 -24066.84,E2 -24066.84} C_VEL
LIN {X 0,Y 170.226,Z 249.287,A -85,B 0,C 180,E1 -24069.992,E2 -24069.992} C_VEL
LIN {X 0,Y 167.377,Z 241.559,A -85,B 0,C 180,E1 -24072.709,E2 -24072.709} C_VEL
LIN {X 0,Y 162.768,Z 231.921,A -85,B 0,C 180,E1 -24076.305,E2 -24076.305} C_VEL
LIN {X 0,Y 158.721,Z 224.811,A -85,B 0,C 180,E1 -24079.225,E2 -24079.225} C_VEL
LIN {X 0,Y 156.182,Z 220.788,A -85,B 0,C 180,E1 -24080.953,E2 -24080.953} C_VEL
LIN {X 0,Y 154.106,Z 217.871,A -85,B 0,C 180,E1 -24082.379,E2 -24082.379} C_VEL
LIN {X 0,Y 153.413,Z 216.34,A -85,B 0,C 180,E1 -24082.962,E2 -24082.962} C_VEL
LIN {X 0,Y 151.266,Z 214.156,A -85,B 0,C 180,E1 -24084.395,E2 -24084.395} C_VEL
LIN {X 0,Y 150.256,Z 211.644,A -85,B 0,C 180,E1 -24085.248,E2 -24085.248} C_VEL
LIN {X 0,Y 150.2,Z 211.276,A -85,B 0,C 180,E1 -24085.437,E2 -24085.437} C_VEL
LIN {X 0,Y 150.204,Z 211.273,A -85,B 0,C 180,E1 -24089.025,E2 -24089.025} C_VEL
LIN {X 0,Y 150.239,Z 211.272,A -85,B 0,C 180,E1 -24092.721,E2 -24092.721} C_VEL
LIN {X 0,Y 150.348,Z 211.248,A -85,B 0,C 180,E1 -24099.209,E2 -24099.209} C_VEL
LIN {X 0,Y 150.351,Z 211.252,A -85,B 0,C 180,E1 -24103.714,E2 -24103.714} C_VEL
LIN {X 0,Y 150.609,Z 211.218,A -85,B 0,C 180,E1 -24109.244,E2 -24109.244} C_VEL
LIN {X 0,Y 150.702,Z 211.211,A -85,B 0,C 180,E1 -24111.959,E2 -24111.959} C_VEL
LIN {X 0,Y 151.215,Z 211.119,A -85,B 0,C 180,E1 -24120.001,E2 -24120.001} C_VEL
LIN {X 0,Y 150.703,Z 211.214,A -85,B 0,C 180,E1 -24128.044,E2 -24128.044} C_VEL
LIN {X 0,Y 150.577,Z 211.23,A -85,B 0,C 180,E1 -24131.439,E2 -24131.439} C_VEL
LIN {X 0,Y 150.352,Z 211.257,A -85,B 0,C 180,E1 -24136.289,E2 -24136.289} C_VEL
LIN {X 0,Y 150.405,Z 211.906,A -85,B 0,C 180,E1 -24140.848,E2 -24140.848} C_VEL
LIN {X 0,Y 150.487,Z 212.88,A -85,B 0,C 180,E1 -24144.856,E2 -24144.856} C_VEL
LIN {X 0,Y 150.585,Z 213.665,A -85,B 0,C 180,E1 -24147.823,E2 -24147.823} C_VEL
LIN {X 0,Y 150.735,Z 215.197,A -85,B 0,C 180,E1 -24152.941,E2 -24152.941} C_VEL
LIN {X 0,Y 150.839,Z 216.067,A -85,B 0,C 180,E1 -24155.009,E2 -24155.009} C_VEL
LIN {X 0,Y 152.061,Z 219.298,A -85,B 0,C 180,E1 -24156.005,E2 -24156.005} C_VEL
LIN {X 0,Y 154.3,Z 222.235,A -85,B 0,C 180,E1 -24157.526,E2 -24157.526} C_VEL
LIN {X 0,Y 156.267,Z 226.235,A -85,B 0,C 180,E1 -24159.025,E2 -24159.025} C_VEL
LIN {X 0,Y 157.212,Z 227.877,A -85,B 0,C 180,E1 -24159.676,E2 -24159.676} C_VEL
LIN {X 0,Y 160.953,Z 236.162,A -85,B 0,C 180,E1 -24162.595,E2 -24162.595} C_VEL
LIN {X 0,Y 163.446,Z 244.373,A -85,B 0,C 180,E1 -24165.085,E2 -24165.085} C_VEL
LIN {X 0,Y 165.082,Z 253.672,A -85,B 0,C 180,E1 -24167.706,E2 -24167.706} C_VEL
LIN {X 0,Y 165.852,Z 262.234,A -85,B 0,C 180,E1 -24170.15,E2 -24170.15} C_VEL
LIN {X 0,Y 165.916,Z 271.267,A -85,B 0,C 180,E1 -24172.872,E2 -24172.872} C_VEL
LIN {X 0,Y 165.442,Z 278.347,A -85,B 0,C 180,E1 -24175.157,E2 -24175.157} C_VEL
LIN {X 0,Y 164.652,Z 283.77,A -85,B 0,C 180,E1 -24177.029,E2 -24177.029} C_VEL
LIN {X 0,Y 161.963,Z 290.414,A -85,B 0,C 180,E1 -24179.346,E2 -24179.346} C_VEL
LIN {X 0,Y 158.397,Z 298.074,A -85,B 0,C 180,E1 -24182.55,E2 -24182.55} C_VEL
LIN {X 0,Y 155.277,Z 304.408,A -85,B 0,C 180,E1 -24185.962,E2 -24185.962} C_VEL
LIN {X 0,Y 152.452,Z 309.904,A -85,B 0,C 180,E1 -24189.773,E2 -24189.773} C_VEL
LIN {X 0,Y 150.231,Z 314.233,A -85,B 0,C 180,E1 -24193.699,E2 -24193.699} C_VEL
LIN {X 0,Y 149.221,Z 316.607,A -85,B 0,C 180,E1 -24196.38,E2 -24196.38} C_VEL
LIN {X 0,Y 148.44,Z 318.413,A -85,B 0,C 180,E1 -24199.083,E2 -24199.083} C_VEL
LIN {X 0,Y 147.692,Z 320.875,A -85,B 0,C 180,E1 -24204.539,E2 -24204.539} C_VEL
LIN {X 0,Y 147.628,Z 321.627,A -85,B 0,C 180,E1 -24208.722,E2 -24208.722} C_VEL
LIN {X 0,Y 147.613,Z 321.471,A -85,B 0,C 180,E1 -24212.729,E2 -24212.729} C_VEL
LIN {X 0,Y 147.692,Z 320.875,A -85,B 0,C 180,E1 -24215.461,E2 -24215.461} C_VEL
LIN {X 0,Y 148.441,Z 318.413,A -85,B 0,C 180,E1 -24220.917,E2 -24220.917} C_VEL
LIN {X 0,Y 149.703,Z 315.454,A -85,B 0,C 180,E1 -24224.963,E2 -24224.963} C_VEL
LIN {X 0,Y 151.623,Z 311.459,A -85,B 0,C 180,E1 -24228.933,E2 -24228.933} C_VEL
LIN {X 0,Y 154.27,Z 306.325,A -85,B 0,C 180,E1 -24232.782,E2 -24232.782} C_VEL
LIN {X 0,Y 156.993,Z 301.063,A -85,B 0,C 180,E1 -24235.879,E2 -24235.879} C_VEL
LIN {X 0,Y 159.169,Z 296.351,A -85,B 0,C 180,E1 -24238.214,E2 -24238.214} C_VEL
LIN {X 0,Y 161.939,Z 290.413,A -85,B 0,C 180,E1 -24240.659,E2 -24240.659} C_VEL
LIN {X 0,Y 164.125,Z 285.531,A -85,B 0,C 180,E1 -24242.361,E2 -24242.361} C_VEL
LIN {X 0,Y 164.982,Z 281.835,A -85,B 0,C 180,E1 -24243.626,E2 -24243.626} C_VEL
LIN {X 0,Y 165.814,Z 273.565,A -85,B 0,C 180,E1 -24246.397,E2 -24246.397} C_VEL
LIN {X 0,Y 165.968,Z 266.311,A -85,B 0,C 180,E1 -24248.652,E2 -24248.652} C_VEL
LIN {X 0,Y 165.53,Z 257.991,A -85,B 0,C 180,E1 -24251.094,E2 -24251.094} C_VEL
LIN {X 0,Y 164.239,Z 248.388,A -85,B 0,C 180,E1 -24253.804,E2 -24253.804} C_VEL
LIN {X 0,Y 162.36,Z 240.263,A -85,B 0,C 180,E1 -24256.163,E2 -24256.163} C_VEL
LIN {X 0,Y 159.49,Z 232.571,A -85,B 0,C 180,E1 -24258.623,E2 -24258.623} C_VEL
LIN {X 0,Y 157.037,Z 227.323,A -85,B 0,C 180,E1 -24260.479,E2 -24260.479} C_VEL
LIN {X 0,Y 154.634,Z 223.156,A -85,B 0,C 180,E1 -24262.176,E2 -24262.176} C_VEL
LIN {X 0,Y 153.981,Z 221.57,A -85,B 0,C 180,E1 -24262.728,E2 -24262.728} C_VEL
LIN {X 0,Y 151.402,Z 219.569,A -85,B 0,C 180,E1 -24264.385,E2 -24264.385} C_VEL
LIN {X 0,Y 145.957,Z 216.331,A -85,B 0,C 180,E1 -24267.755,E2 -24267.755} C_VEL
LIN {X 0,Y 143.593,Z 215.404,A -85,B 0,C 180,E1 -24269.491,E2 -24269.491} C_VEL
LIN {X 0,Y 143.462,Z 214.269,A -85,B 0,C 180,E1 -24273.837,E2 -24273.837} C_VEL
LIN {X 0,Y 143.38,Z 212.855,A -85,B 0,C 180,E1 -24279.932,E2 -24279.932} C_VEL
LIN {X 0,Y 143.301,Z 212.265,A -85,B 0,C 180,E1 -24282.885,E2 -24282.885} C_VEL
LIN {X 0,Y 143.536,Z 212.106,A -85,B 0,C 180,E1 -24288.704,E2 -24288.704} C_VEL
LIN {X 0,Y 143.625,Z 212.095,A -85,B 0,C 180,E1 -24291.557,E2 -24291.557} C_VEL
LIN {X 0,Y 144.174,Z 211.994,A -85,B 0,C 180,E1 -24299.998,E2 -24299.998} C_VEL
LIN {X 0,Y 143.623,Z 212.09,A -85,B 0,C 180,E1 -24308.44,E2 -24308.44} C_VEL
LIN {X 0,Y 143.503,Z 212.108,A -85,B 0,C 180,E1 -24311.627,E2 -24311.627} C_VEL
LIN {X 0,Y 143.294,Z 212.136,A -85,B 0,C 180,E1 -24317.113,E2 -24317.113} C_VEL
LIN {X 0,Y 143.274,Z 212.131,A -85,B 0,C 180,E1 -24321.253,E2 -24321.253} C_VEL
LIN {X 0,Y 143.186,Z 212.149,A -85,B 0,C 180,E1 -24327.935,E2 -24327.935} C_VEL
LIN {X 0,Y 143.135,Z 212.155,A -85,B 0,C 180,E1 -24330.419,E2 -24330.419} C_VEL
LIN {X 0,Y 144.059,Z 214.834,A -85,B 0,C 180,E1 -24331.424,E2 -24331.424} C_VEL
LIN {X 0,Y 146.192,Z 217.119,A -85,B 0,C 180,E1 -24333.18,E2 -24333.18} C_VEL
LIN {X 0,Y 147.007,Z 217.994,A -85,B 0,C 180,E1 -24333.827,E2 -24333.827} C_VEL
LIN {X 0,Y 148.649,Z 220.993,A -85,B 0,C 180,E1 -24335.287,E2 -24335.287} C_VEL
LIN {X 0,Y 150.186,Z 222.819,A -85,B 0,C 180,E1 -24336.419,E2 -24336.419} C_VEL
LIN {X 0,Y 152.002,Z 225.903,A -85,B 0,C 180,E1 -24337.905,E2 -24337.905} C_VEL
LIN {X 0,Y 156.699,Z 233.952,A -85,B 0,C 180,E1 -24341.665,E2 -24341.665} C_VEL
LIN {X 0,Y 161.453,Z 244.074,A -85,B 0,C 180,E1 -24345.856,E2 -24345.856} C_VEL
LIN {X 0,Y 164.724,Z 253.491,A -85,B 0,C 180,E1 -24349.457,E2 -24349.457} C_VEL
LIN {X 0,Y 166.891,Z 261.928,A -85,B 0,C 180,E1 -24352.638,E2 -24352.638} C_VEL
LIN {X 0,Y 168.325,Z 270.841,A -85,B 0,C 180,E1 -24356.098,E2 -24356.098} C_VEL
LIN {X 0,Y 169.56,Z 277.091,A -85,B 0,C 180,E1 -24358.797,E2 -24358.797} C_VEL
LIN {X 0,Y 172.136,Z 284.652,A -85,B 0,C 180,E1 -24362.657,E2 -24362.657} C_VEL
LIN {X 0,Y 176.095,Z 291.171,A -85,B 0,C 180,E1 -24366.623,E2 -24366.623} C_VEL
LIN {X 0,Y 179.895,Z 295.552,A -85,B 0,C 180,E1 -24369.65,E2 -24369.65} C_VEL
LIN {X 0,Y 186.355,Z 300.489,A -85,B 0,C 180,E1 -24373.682,E2 -24373.682} C_VEL
LIN {X 0,Y 194.242,Z 304.536,A -85,B 0,C 180,E1 -24377.656,E2 -24377.656} C_VEL
LIN {X 0,Y 199.784,Z 306.605,A -85,B 0,C 180,E1 -24380.051,E2 -24380.051} C_VEL
LIN {X 0,Y 205.62,Z 308.246,A -85,B 0,C 180,E1 -24382.386,E2 -24382.386} C_VEL
LIN {X 0,Y 211.753,Z 309.435,A -85,B 0,C 180,E1 -24384.666,E2 -24384.666} C_VEL
LIN {X 0,Y 218.153,Z 310.28,A -85,B 0,C 180,E1 -24387.049,E2 -24387.049} C_VEL
LIN {X 0,Y 220.832,Z 310.531,A -85,B 0,C 180,E1 -24388.176,E2 -24388.176} C_VEL
LIN {X 0,Y 224.568,Z 310.59,A -85,B 0,C 180,E1 -24390,E2 -24390} C_VEL
LIN {X 0,Y 220.835,Z 310.531,A -85,B 0,C 180,E1 -24391.824,E2 -24391.824} C_VEL
LIN {X 0,Y 216.088,Z 310.104,A -85,B 0,C 180,E1 -24393.73,E2 -24393.73} C_VEL
LIN {X 0,Y 210.626,Z 309.238,A -85,B 0,C 180,E1 -24395.745,E2 -24395.745} C_VEL
LIN {X 0,Y 204.874,Z 308.064,A -85,B 0,C 180,E1 -24397.887,E2 -24397.887} C_VEL
LIN {X 0,Y 199.194,Z 306.455,A -85,B 0,C 180,E1 -24400.161,E2 -24400.161} C_VEL
LIN {X 0,Y 189.045,Z 302.081,A -85,B 0,C 180,E1 -24404.859,E2 -24404.859} C_VEL
LIN {X 0,Y 183.831,Z 298.798,A -85,B 0,C 180,E1 -24407.809,E2 -24407.809} C_VEL
LIN {X 0,Y 177.575,Z 293.119,A -85,B 0,C 180,E1 -24412.085,E2 -24412.085} C_VEL
LIN {X 0,Y 173.387,Z 287.087,A -85,B 0,C 180,E1 -24415.934,E2 -24415.934} C_VEL
LIN {X 0,Y 170.729,Z 281.116,A -85,B 0,C 180,E1 -24419.224,E2 -24419.224} C_VEL
LIN {X 0,Y 168.739,Z 273.524,A -85,B 0,C 180,E1 -24422.782,E2 -24422.782} C_VEL
LIN {X 0,Y 167.543,Z 265.557,A -85,B 0,C 180,E1 -24425.962,E2 -24425.962} C_VEL
LIN {X 0,Y 166.161,Z 258.873,A -85,B 0,C 180,E1 -24428.516,E2 -24428.516} C_VEL
LIN {X 0,Y 163.875,Z 250.93,A -85,B 0,C 180,E1 -24431.525,E2 -24431.525} C_VEL
LIN {X 0,Y 160.884,Z 242.686,A -85,B 0,C 180,E1 -24434.691,E2 -24434.691} C_VEL
LIN {X 0,Y 156.683,Z 233.955,A -85,B 0,C 180,E1 -24438.342,E2 -24438.342} C_VEL
LIN {X 0,Y 151.99,Z 225.923,A -85,B 0,C 180,E1 -24442.097,E2 -24442.097} C_VEL
LIN {X 0,Y 149.59,Z 221.963,A -85,B 0,C 180,E1 -24444.038,E2 -24444.038} C_VEL
LIN {X 0,Y 147.46,Z 219.136,A -85,B 0,C 180,E1 -24445.706,E2 -24445.706} C_VEL
LIN {X 0,Y 146.671,Z 217.423,A -85,B 0,C 180,E1 -24446.475,E2 -24446.475} C_VEL
LIN {X 0,Y 144.33,Z 215.24,A -85,B 0,C 180,E1 -24448.335,E2 -24448.335} C_VEL
LIN {X 0,Y 143.263,Z 212.775,A -85,B 0,C 180,E1 -24449.407,E2 -24449.407} C_VEL
LIN {X 0,Y 143.139,Z 212.155,A -85,B 0,C 180,E1 -24449.684,E2 -24449.684} C_VEL
LIN {X 0,Y 143.153,Z 212.147,A -85,B 0,C 180,E1 -24453.78,E2 -24453.78} C_VEL
LIN {X 0,Y 143.304,Z 212.124,A -85,B 0,C 180,E1 -24459.924,E2 -24459.924} C_VEL
LIN {X 0,Y 143.351,Z 212.12,A -85,B 0,C 180,E1 -24465.812,E2 -24465.812} C_VEL
LIN {X 0,Y 143.535,Z 212.102,A -85,B 0,C 180,E1 -24468.707,E2 -24468.707} C_VEL
LIN {X 0,Y 143.623,Z 212.09,A -85,B 0,C 180,E1 -24471.56,E2 -24471.56} C_VEL
LIN {X 0,Y 144.174,Z 211.994,A -85,B 0,C 180,E1 -24480.002,E2 -24480.002} C_VEL
LIN {X 0,Y 143.625,Z 212.095,A -85,B 0,C 180,E1 -24488.443,E2 -24488.443} C_VEL
LIN {X 0,Y 143.504,Z 212.112,A -85,B 0,C 180,E1 -24491.63,E2 -24491.63} C_VEL
LIN {X 0,Y 143.301,Z 212.265,A -85,B 0,C 180,E1 -24497.115,E2 -24497.115} C_VEL
LIN {X 0,Y 143.391,Z 213.138,A -85,B 0,C 180,E1 -24501.373,E2 -24501.373} C_VEL
LIN {X 0,Y 143.568,Z 214.834,A -85,B 0,C 180,E1 -24508.221,E2 -24508.221} C_VEL
LIN {X 0,Y 143.67,Z 215.787,A -85,B 0,C 180,E1 -24510.704,E2 -24510.704} C_VEL
LIN {X 0,Y 144.828,Z 218.882,A -85,B 0,C 180,E1 -24511.854,E2 -24511.854} C_VEL
LIN {X 0,Y 147.406,Z 222.104,A -85,B 0,C 180,E1 -24513.922,E2 -24513.922} C_VEL
